// @TEST-ASSERT
AssertTrue(Condition := equal, Message := 'Did not convert DINT to REAL correctly');
AssertTrue(Condition := converted, Message := 'Did not report DINT to REAL conversion was successful');

TEST_FINISHED();
END_METHOD

METHOD PUBLIC Check_DINT_TO_REAL_Max
VAR
	value : DINT := DatatypeLimits.DINT_MAX_VALUE;
	actual : REAL;
	converted : BOOL;
	equal : BOOL;
END_VAR
TEST('Check_DINT_TO_REAL_Max');

// @TEST-RUN
converted := TryConvert_DINT_TO_Destination(value, actual);
equal := actual = DINT_TO_REAL(value);

// @TEST-ASSERT
AssertTrue(Condition := equal, Message := 'Did not convert DINT to REAL correctly');
AssertTrue(Condition := converted, Message := 'Did not report DINT to REAL conversion was successful');

TEST_FINISHED();
END_METHOD

METHOD PUBLIC Check_DINT_TO_SINT_Min
VAR
	value : DINT := DatatypeLimits.MIN_VALUE_OF_DINT_WHICH_CAN_BE_HELD_IN_A_SINT;
	actual : SINT;
	converted : BOOL;
	equal : BOOL;
END_VAR
TEST('Check_DINT_TO_SINT_Min');

// @TEST-RUN
converted := TryConvert_DINT_TO_Destination(value, actual);
equal := actual = DINT_TO_SINT(value);

// @TEST-ASSERT
AssertTrue(Condition := equal, Message := 'Did not convert DINT to SINT correctly');
AssertTrue(Condition := converted, Message := 'Did not report DINT to SINT conversion was successful');

TEST_FINISHED();
END_METHOD

METHOD PUBLIC Check_DINT_TO_SINT_TooHigh
VAR
	value : DINT := DatatypeLimits.DINT_MAX_VALUE;
	actual : SINT;
	converted : BOOL;
END_VAR
TEST('Check_DINT_TO_SINT_TooHigh');

// @TEST-RUN
converted := TryConvert_DINT_TO_Destination(value, actual);

// @TEST-ASSERT
AssertFalse(Condition := converted, Message := 'Did not report DINT to SINT conversion was prevented');

TEST_FINISHED();
END_METHOD

METHOD PUBLIC Check_DINT_TO_SINT_TooLow
VAR
	value : DINT := DatatypeLimits.DINT_MIN_VALUE;
	actual : SINT;
	converted : BOOL;
END_VAR
TEST('Check_DINT_TO_SINT_TooLow');

// @TEST-RUN
converted := TryConvert_DINT_TO_Destination(value, actual);

// @TEST-ASSERT
AssertFalse(Condition := converted, Message := 'Did not report DINT to SINT conversion was prevented');

TEST_FINISHED();
END_METHOD

METHOD PUBLIC Check_DINT_TO_SINT_Max
VAR
	value : DINT := DatatypeLimits.MAX_VALUE_OF_DINT_WHICH_CAN_BE_HELD_IN_A_SINT;
	actual : SINT;
	converted : BOOL;
	equal : BOOL;
END_VAR
TEST('Check_DINT_TO_SINT_Max');

// @TEST-RUN
converted := TryConvert_DINT_TO_Destination(value, actual);
equal := actual = DINT_TO_SINT(value);

// @TEST-ASSERT
AssertTrue(Condition := equal, Message := 'Did not convert DINT to SINT correctly');
AssertTrue(Condition := converted, Message := 'Did not report DINT to SINT conversion was successful');

TEST_FINISHED();
END_METHOD

METHOD PUBLIC Check_DINT_TO_STRING_Min
VAR
	value : DINT := DatatypeLimits.DINT_MIN_VALUE;
	actual : STRING;
	converted : BOOL;
	equal : BOOL;
END_VAR
TEST('Check_DINT_TO_STRING_Min');

// @TEST-RUN
converted := TryConvert_DINT_TO_Destination(value, actual);
equal := actual = DINT_TO_STRING(value);

// @TEST-ASSERT
AssertTrue(Condition := equal, Message := 'Did not convert DINT to STRING correctly');
AssertTrue(Condition := converted, Message := 'Did not report DINT to STRING conversion was successful');

TEST_FINISHED();
END_METHOD

METHOD PUBLIC Check_DINT_TO_STRING_Max
VAR
	value : DINT := DatatypeLimits.DINT_MAX_VALUE;
	actual : STRING;
	converted : BOOL;
	equal : BOOL;
END_VAR
TEST('Check_DINT_TO_STRING_Max');

// @TEST-RUN
converted := TryConvert_DINT_TO_Destination(value, actual);
equal := actual = DINT_TO_STRING(value);

// @TEST-ASSERT
AssertTrue(Condition := equal, Message := 'Did not convert DINT to STRING correctly');
AssertTrue(Condition := converted, Message := 'Did not report DINT to STRING conversion was successful');

TEST_FINISHED();
END_METHOD

METHOD PUBLIC Check_DINT_TO_TIME_Min
VAR
	value : DINT := DatatypeLimits.MIN_VALUE_OF_DINT_WHICH_CAN_BE_HELD_IN_A_TIME;
	actual : TIME;
	converted : BOOL;
	equal : BOOL;
END_VAR
TEST('Check_DINT_TO_TIME_Min');

// @TEST-RUN
converted := TryConvert_DINT_TO_Destination(value, actual);
equal := actual = DINT_TO_TIME(value);

// @TEST-ASSERT
AssertTrue(Condition := equal, Message := 'Did not convert DINT to TIME correctly');
AssertTrue(Condition := converted, Message := 'Did not report DINT to TIME conversion was successful');

TEST_FINISHED();
END_METHOD

METHOD PUBLIC Check_DINT_TO_TIME_TooLow
VAR
	value : DINT := DatatypeLimits.DINT_MIN_VALUE;
	actual : TIME;
	converted : BOOL;
END_VAR
TEST('Check_DINT_TO_TIME_TooLow');

// @TEST-RUN
converted := TryConvert_DINT_TO_Destination(value, actual);

// @TEST-ASSERT
AssertFalse(Condition := converted, Message := 'Did not report DINT to TIME conversion was prevented');

TEST_FINISHED();
END_METHOD

METHOD PUBLIC Check_DINT_TO_TIME_Max
VAR
	value : DINT := DatatypeLimits.DINT_MAX_VALUE;
	actual : TIME;
	converted : BOOL;
	equal : BOOL;
END_VAR
TEST('Check_DINT_TO_TIME_Max');

// @TEST-RUN
converted := TryConvert_DINT_TO_Destination(value, actual);
equal := actual = DINT_TO_TIME(value);

// @TEST-ASSERT
AssertTrue(Condition := equal, Message := 'Did not convert DINT to TIME correctly');
AssertTrue(Condition := converted, Message := 'Did not report DINT to TIME conversion was successful');

TEST_FINISHED();
END_METHOD

METHOD PUBLIC Check_DINT_TO_TOD_Min
VAR
	value : DINT := DatatypeLimits.MIN_VALUE_OF_DINT_WHICH_CAN_BE_HELD_IN_A_TOD;
	actual : TOD;
	converted : BOOL;
	equal : BOOL;
END_VAR
TEST('Check_DINT_TO_TOD_Min');

// @TEST-RUN
converted := TryConvert_DINT_TO_Destination(value, actual);
equal := actual = DINT_TO_TOD(value);

// @TEST-ASSERT
AssertTrue(Condition := equal, Message := 'Did not convert DINT to TOD correctly');
AssertTrue(Condition := converted, Message := 'Did not report DINT to TOD conversion was successful');

TEST_FINISHED();
END_METHOD

METHOD PUBLIC Check_DINT_TO_TOD_TooHigh
VAR
	value : DINT := DatatypeLimits.DINT_MAX_VALUE;
	actual : TOD;
	converted : BOOL;
END_VAR
TEST('Check_DINT_TO_TOD_TooHigh');

// @TEST-RUN
converted := TryConvert_DINT_TO_Destination(value, actual);

// @TEST-ASSERT
AssertFalse(Condition := converted, Message := 'Did not report DINT to TOD conversion was prevented');

TEST_FINISHED();
END_METHOD

METHOD PUBLIC Check_DINT_TO_TOD_TooLow
VAR
	value : DINT := DatatypeLimits.DINT_MIN_VALUE;
	actual : TOD;
	converted : BOOL;
END_VAR
TEST('Check_DINT_TO_TOD_TooLow');

// @TEST-RUN
converted := TryConvert_DINT_TO_Destination(value, actual);

// @TEST-ASSERT
AssertFalse(Condition := converted, Message := 'Did not report DINT to TOD conversion was prevented');

TEST_FINISHED();
END_METHOD

METHOD PUBLIC Check_DINT_TO_TOD_Max
VAR
	value : DINT := DatatypeLimits.MAX_VALUE_OF_DINT_WHICH_CAN_BE_HELD_IN_A_TOD;
	actual : TOD;
	converted : BOOL;
	equal : BOOL;
END_VAR
TEST('Check_DINT_TO_TOD_Max');

// @TEST-RUN
converted := TryConvert_DINT_TO_Destination(value, actual);
equal := actual = DINT_TO_TOD(value);

// @TEST-ASSERT
AssertTrue(Condition := equal, Message := 'Did not convert DINT to TOD correctly');
AssertTrue(Condition := converted, Message := 'Did not report DINT to TOD conversion was successful');

TEST_FINISHED();
END_METHOD

METHOD PUBLIC Check_DINT_TO_UDINT_Min
VAR
	value : DINT := DatatypeLimits.MIN_VALUE_OF_DINT_WHICH_CAN_BE_HELD_IN_A_UDINT;
	actual : UDINT;
	converted : BOOL;
	equal : BOOL;
END_VAR
TEST('Check_DINT_TO_UDINT_Min');

// @TEST-RUN
converted := TryConvert_DINT_TO_Destination(value, actual);
equal := actual = DINT_TO_UDINT(value);

// @TEST-ASSERT
AssertTrue(Condition := equal, Message := 'Did not convert DINT to UDINT correctly');
AssertTrue(Condition := converted, Message := 'Did not report DINT to UDINT conversion was successful');

TEST_FINISHED();
END_METHOD

METHOD PUBLIC Check_DINT_TO_UDINT_TooLow
VAR
	value : DINT := DatatypeLimits.DINT_MIN_VALUE;
	actual : UDINT;
	converted : BOOL;
END_VAR
TEST('Check_DINT_TO_UDINT_TooLow');

// @TEST-RUN
converted := TryConvert_DINT_TO_Destination(value, actual);

// @TEST-ASSERT
AssertFalse(Condition := converted, Message := 'Did not report DINT to UDINT conversion was prevented');

TEST_FINISHED();
END_METHOD

METHOD PUBLIC Check_DINT_TO_UDINT_Max
VAR
	value : DINT := DatatypeLimits.DINT_MAX_VALUE;
	actual : UDINT;
	converted : BOOL;
	equal : BOOL;
END_VAR
TEST('Check_DINT_TO_UDINT_Max');

// @TEST-RUN
converted := TryConvert_DINT_TO_Destination(value, actual);
equal := actual = DINT_TO_UDINT(value);

// @TEST-ASSERT
AssertTrue(Condition := equal, Message := 'Did not convert DINT to UDINT correctly');
AssertTrue(Condition := converted, Message := 'Did not report DINT to UDINT conversion was successful');

TEST_FINISHED();
END_METHOD

METHOD PUBLIC Check_DINT_TO_UINT_Min
VAR
	value : DINT := DatatypeLimits.MIN_VALUE_OF_DINT_WHICH_CAN_BE_HELD_IN_A_UINT;
	actual : UINT;
	converted : BOOL;
	equal : BOOL;
END_VAR
TEST('Check_DINT_TO_UINT_Min');

// @TEST-RUN
converted := TryConvert_DINT_TO_Destination(value, actual);
equal := actual = DINT_TO_UINT(value);

// @TEST-ASSERT
AssertTrue(Condition := equal, Message := 'Did not convert DINT to UINT correctly');
AssertTrue(Condition := converted, Message := 'Did not report DINT to UINT conversion was successful');

TEST_FINISHED();
END_METHOD

METHOD PUBLIC Check_DINT_TO_UINT_TooHigh
VAR
	value : DINT := DatatypeLimits.DINT_MAX_VALUE;
	actual : UINT;
	converted : BOOL;
END_VAR
TEST('Check_DINT_TO_UINT_TooHigh');

// @TEST-RUN
converted := TryConvert_DINT_TO_Destination(value, actual);

// @TEST-ASSERT
AssertFalse(Condition := converted, Message := 'Did not report DINT to UINT conversion was prevented');

TEST_FINISHED();
END_METHOD

METHOD PUBLIC Check_DINT_TO_UINT_TooLow
VAR
	value : DINT := DatatypeLimits.DINT_MIN_VALUE;
	actual : UINT;
	converted : BOOL;
END_VAR
TEST('Check_DINT_TO_UINT_TooLow');

// @TEST-RUN
converted := TryConvert_DINT_TO_Destination(value, actual);

// @TEST-ASSERT
AssertFalse(Condition := converted, Message := 'Did not report DINT to UINT conversion was prevented');

TEST_FINISHED();
END_METHOD

METHOD PUBLIC Check_DINT_TO_UINT_Max
VAR
	value : DINT := DatatypeLimits.MAX_VALUE_OF_DINT_WHICH_CAN_BE_HELD_IN_A_UINT;
	actual : UINT;
	converted : BOOL;
	equal : BOOL;
END_VAR
TEST('Check_DINT_TO_UINT_Max');

// @TEST-RUN
converted := TryConvert_DINT_TO_Destination(value, actual);
equal := actual = DINT_TO_UINT(value);

// @TEST-ASSERT
AssertTrue(Condition := equal, Message := 'Did not convert DINT to UINT correctly');
AssertTrue(Condition := converted, Message := 'Did not report DINT to UINT conversion was successful');

TEST_FINISHED();
END_METHOD

METHOD PUBLIC Check_DINT_TO_ULINT_Min
VAR
	value : DINT := DatatypeLimits.MIN_VALUE_OF_DINT_WHICH_CAN_BE_HELD_IN_A_ULINT;
	actual : ULINT;
	converted : BOOL;
	equal : BOOL;
END_VAR
TEST('Check_DINT_TO_ULINT_Min');

// @TEST-RUN
converted := TryConvert_DINT_TO_Destination(value, actual);
equal := actual = DINT_TO_ULINT(value);

// @TEST-ASSERT
AssertTrue(Condition := equal, Message := 'Did not convert DINT to ULINT correctly');
AssertTrue(Condition := converted, Message := 'Did not report DINT to ULINT conversion was successful');

TEST_FINISHED();
END_METHOD

METHOD PUBLIC Check_DINT_TO_ULINT_TooLow
VAR
	value : DINT := DatatypeLimits.DINT_MIN_VALUE;
	actual : ULINT;
	converted : BOOL;
END_VAR
TEST('Check_DINT_TO_ULINT_TooLow');

// @TEST-RUN
converted := TryConvert_DINT_TO_Destination(value, actual);

// @TEST-ASSERT
AssertFalse(Condition := converted, Message := 'Did not report DINT to ULINT conversion was prevented');

TEST_FINISHED();
END_METHOD

METHOD PUBLIC Check_DINT_TO_ULINT_Max
VAR
	value : DINT := DatatypeLimits.DINT_MAX_VALUE;
	actual : ULINT;
	converted : BOOL;
	equal : BOOL;
END_VAR
TEST('Check_DINT_TO_ULINT_Max');

// @TEST-RUN
converted := TryConvert_DINT_TO_Destination(value, actual);
equal := actual = DINT_TO_ULINT(value);

// @TEST-ASSERT
AssertTrue(Condition := equal, Message := 'Did not convert DINT to ULINT correctly');
AssertTrue(Condition := converted, Message := 'Did not report DINT to ULINT conversion was successful');

TEST_FINISHED();
END_METHOD

METHOD PUBLIC Check_DINT_TO_USINT_Min
VAR
	value : DINT := DatatypeLimits.MIN_VALUE_OF_DINT_WHICH_CAN_BE_HELD_IN_A_USINT;
	actual : USINT;
	converted : BOOL;
	equal : BOOL;
END_VAR
TEST('Check_DINT_TO_USINT_Min');

// @TEST-RUN
converted := TryConvert_DINT_TO_Destination(value, actual);
equal := actual = DINT_TO_USINT(value);

// @TEST-ASSERT
AssertTrue(Condition := equal, Message := 'Did not convert DINT to USINT correctly');
AssertTrue(Condition := converted, Message := 'Did not report DINT to USINT conversion was successful');

TEST_FINISHED();
END_METHOD

METHOD PUBLIC Check_DINT_TO_USINT_TooHigh
VAR
	value : DINT := DatatypeLimits.DINT_MAX_VALUE;
	actual : USINT;
	converted : BOOL;
END_VAR
TEST('Check_DINT_TO_USINT_TooHigh');

// @TEST-RUN
converted := TryConvert_DINT_TO_Destination(value, actual);

// @TEST-ASSERT
AssertFalse(Condition := converted, Message := 'Did not report DINT to USINT conversion was prevented');

TEST_FINISHED();
END_METHOD

METHOD PUBLIC Check_DINT_TO_USINT_TooLow
VAR
	value : DINT := DatatypeLimits.DINT_MIN_VALUE;
	actual : USINT;
	converted : BOOL;
END_VAR
TEST('Check_DINT_TO_USINT_TooLow');

// @TEST-RUN
converted := TryConvert_DINT_TO_Destination(value, actual);

// @TEST-ASSERT
AssertFalse(Condition := converted, Message := 'Did not report DINT to USINT conversion was prevented');

TEST_FINISHED();
END_METHOD

METHOD PUBLIC Check_DINT_TO_USINT_Max
VAR
	value : DINT := DatatypeLimits.MAX_VALUE_OF_DINT_WHICH_CAN_BE_HELD_IN_A_USINT;
	actual : USINT;
	converted : BOOL;
	equal : BOOL;
END_VAR
TEST('Check_DINT_TO_USINT_Max');

// @TEST-RUN
converted := TryConvert_DINT_TO_Destination(value, actual);
equal := actual = DINT_TO_USINT(value);

// @TEST-ASSERT
AssertTrue(Condition := equal, Message := 'Did not convert DINT to USINT correctly');
AssertTrue(Condition := converted, Message := 'Did not report DINT to USINT conversion was successful');

TEST_FINISHED();
END_METHOD

METHOD PUBLIC Check_DINT_TO_WORD_Min
VAR
	value : DINT := DatatypeLimits.MIN_VALUE_OF_DINT_WHICH_CAN_BE_HELD_IN_A_WORD;
	actual : WORD;
	converted : BOOL;
	equal : BOOL;
END_VAR
TEST('Check_DINT_TO_WORD_Min');

// @TEST-RUN
converted := TryConvert_DINT_TO_Destination(value, actual);
equal := actual = DINT_TO_WORD(value);

// @TEST-ASSERT
AssertTrue(Condition := equal, Message := 'Did not convert DINT to WORD correctly');
AssertTrue(Condition := converted, Message := 'Did not report DINT to WORD conversion was successful');

TEST_FINISHED();
END_METHOD

METHOD PUBLIC Check_DINT_TO_WORD_TooHigh
VAR
	value : DINT := DatatypeLimits.DINT_MAX_VALUE;
	actual : WORD;
	converted : BOOL;
END_VAR
TEST('Check_DINT_TO_WORD_TooHigh');

// @TEST-RUN
converted := TryConvert_DINT_TO_Destination(value, actual);

// @TEST-ASSERT
AssertFalse(Condition := converted, Message := 'Did not report DINT to WORD conversion was prevented');

TEST_FINISHED();
END_METHOD

METHOD PUBLIC Check_DINT_TO_WORD_TooLow
VAR
	value : DINT := DatatypeLimits.DINT_MIN_VALUE;
	actual : WORD;
	converted : BOOL;
END_VAR
TEST('Check_DINT_TO_WORD_TooLow');

// @TEST-RUN
converted := TryConvert_DINT_TO_Destination(value, actual);

// @TEST-ASSERT
AssertFalse(Condition := converted, Message := 'Did not report DINT to WORD conversion was prevented');

TEST_FINISHED();
END_METHOD

METHOD PUBLIC Check_DINT_TO_WORD_Max
VAR
	value : DINT := DatatypeLimits.MAX_VALUE_OF_DINT_WHICH_CAN_BE_HELD_IN_A_WORD;
	actual : WORD;
	converted : BOOL;
	equal : BOOL;
END_VAR
TEST('Check_DINT_TO_WORD_Max');

// @TEST-RUN
converted := TryConvert_DINT_TO_Destination(value, actual);
equal := actual = DINT_TO_WORD(value);

// @TEST-ASSERT
AssertTrue(Condition := equal, Message := 'Did not convert DINT to WORD correctly');
AssertTrue(Condition := converted, Message := 'Did not report DINT to WORD conversion was successful');

TEST_FINISHED();
END_METHOD

END_FUNCTION_BLOCK

// ---- Tests/LINT_TO_TestSuite.TcPOU
FUNCTION_BLOCK PUBLIC LINT_TO_TestSuite EXTENDS TcUnit.FB_TestSuite
VAR
END_VAR

Check_LINT_TO_BOOL_Max();
Check_LINT_TO_BOOL_Min();
Check_LINT_TO_BYTE_Max();
Check_LINT_TO_BYTE_Min();
Check_LINT_TO_BYTE_TooHigh();
Check_LINT_TO_BYTE_TooLow();
Check_LINT_TO_WORD_Max();
Check_LINT_TO_WORD_Min();
Check_LINT_TO_WORD_TooHigh();
Check_LINT_TO_WORD_TooLow();
Check_LINT_TO_DWORD_Max();
Check_LINT_TO_DWORD_Min();
Check_LINT_TO_DWORD_TooHigh();
Check_LINT_TO_DWORD_TooLow();
Check_LINT_TO_LWORD_Max();
Check_LINT_TO_LWORD_Min();
Check_LINT_TO_LWORD_TooLow();
Check_LINT_TO_SINT_Max();
Check_LINT_TO_SINT_Min();
Check_LINT_TO_SINT_TooHigh();
Check_LINT_TO_SINT_TooLow();
Check_LINT_TO_INT_Max();
Check_LINT_TO_INT_Min();
Check_LINT_TO_INT_TooHigh();
Check_LINT_TO_INT_TooLow();
Check_LINT_TO_DINT_Max();
Check_LINT_TO_DINT_Min();
Check_LINT_TO_DINT_TooHigh();
Check_LINT_TO_DINT_TooLow();
Check_LINT_TO_LINT_Max();
Check_LINT_TO_LINT_Min();
Check_LINT_TO_USINT_Max();
Check_LINT_TO_USINT_Min();
Check_LINT_TO_USINT_TooHigh();
Check_LINT_TO_USINT_TooLow();
Check_LINT_TO_UINT_Max();
Check_LINT_TO_UINT_Min();
Check_LINT_TO_UINT_TooHigh();
Check_LINT_TO_UINT_TooLow();
Check_LINT_TO_UDINT_Max();
Check_LINT_TO_UDINT_Min();
Check_LINT_TO_UDINT_TooHigh();
Check_LINT_TO_UDINT_TooLow();
Check_LINT_TO_ULINT_Max();
Check_LINT_TO_ULINT_Min();
Check_LINT_TO_ULINT_TooLow();
Check_LINT_TO_REAL_Max();
Check_LINT_TO_REAL_Min();
Check_LINT_TO_LREAL_Max();
Check_LINT_TO_LREAL_Min();
Check_LINT_TO_TIME_Max();
Check_LINT_TO_TIME_Min();
Check_LINT_TO_TIME_TooHigh();
Check_LINT_TO_TIME_TooLow();
Check_LINT_TO_TOD_Max();
Check_LINT_TO_TOD_Min();
Check_LINT_TO_TOD_TooHigh();
Check_LINT_TO_TOD_TooLow();
Check_LINT_TO_DATE_Max();
Check_LINT_TO_DATE_Min();
Check_LINT_TO_DATE_TooHigh();
Check_LINT_TO_DATE_TooLow();
Check_LINT_TO_DT_Max();
Check_LINT_TO_DT_Min();
Check_LINT_TO_DT_TooHigh();
Check_LINT_TO_DT_TooLow();
Check_LINT_TO_STRING_Max();
Check_LINT_TO_STRING_Min();

METHOD PUBLIC Check_LINT_TO_BOOL_Min
VAR
	value : LINT := DatatypeLimits.LINT_MIN_VALUE;
	actual : BOOL;
	converted : BOOL;
	equal : BOOL;
END_VAR
TEST('Check_LINT_TO_BOOL_Min');

// @TEST-RUN
converted := TryConvert_LINT_TO_Destination(value, actual);
equal := actual = LINT_TO_BOOL(value);

// @TEST-ASSERT
AssertTrue(Condition := equal, Message := 'Did not convert LINT to BOOL correctly');
AssertTrue(Condition := converted, Message := 'Did not report LINT to BOOL conversion was successful');

TEST_FINISHED();
END_METHOD

METHOD PUBLIC Check_LINT_TO_BOOL_Max
VAR
	value : LINT := DatatypeLimits.LINT_MAX_VALUE;
	actual : BOOL;
	converted : BOOL;
	equal : BOOL;
END_VAR
TEST('Check_LINT_TO_BOOL_Max');

// @TEST-RUN
converted := TryConvert_LINT_TO_Destination(value, actual);
equal := actual = LINT_TO_BOOL(value);

// @TEST-ASSERT
AssertTrue(Condition := equal, Message := 'Did not convert LINT to BOOL correctly');
AssertTrue(Condition := converted, Message := 'Did not report LINT to BOOL conversion was successful');

TEST_FINISHED();
END_METHOD

METHOD PUBLIC Check_LINT_TO_BYTE_Min
VAR
	value : LINT := DatatypeLimits.MIN_VALUE_OF_LINT_WHICH_CAN_BE_HELD_IN_A_BYTE;
	actual : BYTE;
	converted : BOOL;
	equal : BOOL;
END_VAR
TEST('Check_LINT_TO_BYTE_Min');

// @TEST-RUN
converted := TryConvert_LINT_TO_Destination(value, actual);
equal := actual = LINT_TO_BYTE(value);

// @TEST-ASSERT
AssertTrue(Condition := equal, Message := 'Did not convert LINT to BYTE correctly');
AssertTrue(Condition := converted, Message := 'Did not report LINT to BYTE conversion was successful');

TEST_FINISHED();
END_METHOD

METHOD PUBLIC Check_LINT_TO_BYTE_TooHigh
VAR
	value : LINT := DatatypeLimits.LINT_MAX_VALUE;
	actual : BYTE;
	converted : BOOL;
END_VAR
TEST('Check_LINT_TO_BYTE_TooHigh');

// @TEST-RUN
converted := TryConvert_LINT_TO_Destination(value, actual);

// @TEST-ASSERT
AssertFalse(Condition := converted, Message := 'Did not report LINT to BYTE conversion was prevented');

TEST_FINISHED();
END_METHOD

METHOD PUBLIC Check_LINT_TO_BYTE_TooLow
VAR
	value : LINT := DatatypeLimits.LINT_MIN_VALUE;
	actual : BYTE;
	converted : BOOL;
END_VAR
TEST('Check_LINT_TO_BYTE_TooLow');

// @TEST-RUN
converted := TryConvert_LINT_TO_Destination(value, actual);

// @TEST-ASSERT
AssertFalse(Condition := converted, Message := 'Did not report LINT to BYTE conversion was prevented');

TEST_FINISHED();
END_METHOD

METHOD PUBLIC Check_LINT_TO_BYTE_Max
VAR
	value : LINT := DatatypeLimits.MAX_VALUE_OF_LINT_WHICH_CAN_BE_HELD_IN_A_BYTE;
	actual : BYTE;
	converted : BOOL;
	equal : BOOL;
END_VAR
TEST('Check_LINT_TO_BYTE_Max');

// @TEST-RUN
converted := TryConvert_LINT_TO_Destination(value, actual);
equal := actual = LINT_TO_BYTE(value);

// @TEST-ASSERT
AssertTrue(Condition := equal, Message := 'Did not convert LINT to BYTE correctly');
AssertTrue(Condition := converted, Message := 'Did not report LINT to BYTE conversion was successful');

TEST_FINISHED();
END_METHOD

METHOD PUBLIC Check_LINT_TO_DATE_Min
VAR
	value : LINT := DatatypeLimits.MIN_VALUE_OF_LINT_WHICH_CAN_BE_HELD_IN_A_DATE;
	actual : DATE;
	converted : BOOL;
	equal : BOOL;
END_VAR
TEST('Check_LINT_TO_DATE_Min');

// @TEST-RUN
converted := TryConvert_LINT_TO_Destination(value, actual);
equal := actual = LINT_TO_DATE(value);

// @TEST-ASSERT
AssertTrue(Condition := equal, Message := 'Did not convert LINT to DATE correctly');
AssertTrue(Condition := converted, Message := 'Did not report LINT to DATE conversion was successful');

TEST_FINISHED();
END_METHOD

METHOD PUBLIC Check_LINT_TO_DATE_TooHigh
VAR
	value : LINT := DatatypeLimits.LINT_MAX_VALUE;
	actual : DATE;
	converted : BOOL;
END_VAR
TEST('Check_LINT_TO_DATE_TooHigh');

// @TEST-RUN
converted := TryConvert_LINT_TO_Destination(value, actual);

// @TEST-ASSERT
AssertFalse(Condition := converted, Message := 'Did not report LINT to DATE conversion was prevented');

TEST_FINISHED();
END_METHOD

METHOD PUBLIC Check_LINT_TO_DATE_TooLow
VAR
	value : LINT := DatatypeLimits.LINT_MIN_VALUE;
	actual : DATE;
	converted : BOOL;
END_VAR
TEST('Check_LINT_TO_DATE_TooLow');

// @TEST-RUN
converted := TryConvert_LINT_TO_Destination(value, actual);

// @TEST-ASSERT
AssertFalse(Condition := converted, Message := 'Did not report LINT to DATE conversion was prevented');

TEST_FINISHED();
END_METHOD

METHOD PUBLIC Check_LINT_TO_DATE_Max
VAR
	value : LINT := DatatypeLimits.MAX_VALUE_OF_LINT_WHICH_CAN_BE_HELD_IN_A_DATE;
	actual : DATE;
	converted : BOOL;
	equal : BOOL;
END_VAR
TEST('Check_LINT_TO_DATE_Max');

// @TEST-RUN
converted := TryConvert_LINT_TO_Destination(value, actual);
equal := actual = LINT_TO_DATE(value);

// @TEST-ASSERT
AssertTrue(Condition := equal, Message := 'Did not convert LINT to DATE correctly');
AssertTrue(Condition := converted, Message := 'Did not report LINT to DATE conversion was successful');

TEST_FINISHED();
END_METHOD

METHOD PUBLIC Check_LINT_TO_DINT_Min
VAR
	value : LINT := DatatypeLimits.MIN_VALUE_OF_LINT_WHICH_CAN_BE_HELD_IN_A_DINT;
	actual : DINT;
	converted : BOOL;
	equal : BOOL;
END_VAR
TEST('Check_LINT_TO_DINT_Min');

// @TEST-RUN
converted := TryConvert_LINT_TO_Destination(value, actual);
equal := actual = LINT_TO_DINT(value);

// @TEST-ASSERT
AssertTrue(Condition := equal, Message := 'Did not convert LINT to DINT correctly');
AssertTrue(Condition := converted, Message := 'Did not report LINT to DINT conversion was successful');

TEST_FINISHED();
END_METHOD

METHOD PUBLIC Check_LINT_TO_DINT_TooHigh
VAR
	value : LINT := DatatypeLimits.LINT_MAX_VALUE;
	actual : DINT;
	converted : BOOL;
END_VAR
TEST('Check_LINT_TO_DINT_TooHigh');

// @TEST-RUN
converted := TryConvert_LINT_TO_Destination(value, actual);

// @TEST-ASSERT
AssertFalse(Condition := converted, Message := 'Did not report LINT to DINT conversion was prevented');

TEST_FINISHED();
END_METHOD

METHOD PUBLIC Check_LINT_TO_DINT_TooLow
VAR
	value : LINT := DatatypeLimits.LINT_MIN_VALUE;
	actual : DINT;
	converted : BOOL;
END_VAR
TEST('Check_LINT_TO_DINT_TooLow');

// @TEST-RUN
converted := TryConvert_LINT_TO_Destination(value, actual);

// @TEST-ASSERT
AssertFalse(Condition := converted, Message := 'Did not report LINT to DINT conversion was prevented');

TEST_FINISHED();
END_METHOD

METHOD PUBLIC Check_LINT_TO_DINT_Max
VAR
	value : LINT := DatatypeLimits.MAX_VALUE_OF_LINT_WHICH_CAN_BE_HELD_IN_A_DINT;
	actual : DINT;
	converted : BOOL;
	equal : BOOL;
END_VAR
TEST('Check_LINT_TO_DINT_Max');

// @TEST-RUN
converted := TryConvert_LINT_TO_Destination(value, actual);
equal := actual = LINT_TO_DINT(value);

// @TEST-ASSERT
AssertTrue(Condition := equal, Message := 'Did not convert LINT to DINT correctly');
AssertTrue(Condition := converted, Message := 'Did not report LINT to DINT conversion was successful');

TEST_FINISHED();
END_METHOD

METHOD PUBLIC Check_LINT_TO_DT_Min
VAR
	value : LINT := DatatypeLimits.MIN_VALUE_OF_LINT_WHICH_CAN_BE_HELD_IN_A_DT;
	actual : DT;
	converted : BOOL;
	equal : BOOL;
END_VAR
TEST('Check_LINT_TO_DT_Min');

// @TEST-RUN
converted := TryConvert_LINT_TO_Destination(value, actual);
equal := actual = LINT_TO_DT(value);

// @TEST-ASSERT
AssertTrue(Condition := equal, Message := 'Did not convert LINT to DT correctly');
AssertTrue(Condition := converted, Message := 'Did not report LINT to DT conversion was successful');

TEST_FINISHED();
END_METHOD

METHOD PUBLIC Check_LINT_TO_DT_TooHigh
VAR
	value : LINT := DatatypeLimits.LINT_MAX_VALUE;
	actual : DT;
	converted : BOOL;
END_VAR
TEST('Check_LINT_TO_DT_TooHigh');

// @TEST-RUN
converted := TryConvert_LINT_TO_Destination(value, actual);

// @TEST-ASSERT
AssertFalse(Condition := converted, Message := 'Did not report LINT to DT conversion was prevented');

TEST_FINISHED();
END_METHOD

METHOD PUBLIC Check_LINT_TO_DT_TooLow
VAR
	value : LINT := DatatypeLimits.LINT_MIN_VALUE;
	actual : DT;
	converted : BOOL;
END_VAR
TEST('Check_LINT_TO_DT_TooLow');

// @TEST-RUN
converted := TryConvert_LINT_TO_Destination(value, actual);

// @TEST-ASSERT
AssertFalse(Condition := converted, Message := 'Did not report LINT to DT conversion was prevented');

TEST_FINISHED();
END_METHOD

METHOD PUBLIC Check_LINT_TO_DT_Max
VAR
	value : LINT := DatatypeLimits.MAX_VALUE_OF_LINT_WHICH_CAN_BE_HELD_IN_A_DT;
	actual : DT;
	converted : BOOL;
	equal : BOOL;
END_VAR
TEST('Check_LINT_TO_DT_Max');

// @TEST-RUN
converted := TryConvert_LINT_TO_Destination(value, actual);
equal := actual = LINT_TO_DT(value);

// @TEST-ASSERT
AssertTrue(Condition := equal, Message := 'Did not convert LINT to DT correctly');
AssertTrue(Condition := converted, Message := 'Did not report LINT to DT conversion was successful');

TEST_FINISHED();
END_METHOD

METHOD PUBLIC Check_LINT_TO_DWORD_Min
VAR
	value : LINT := DatatypeLimits.MIN_VALUE_OF_LINT_WHICH_CAN_BE_HELD_IN_A_DWORD;
	actual : DWORD;
	converted : BOOL;
	equal : BOOL;
END_VAR
TEST('Check_LINT_TO_DWORD_Min');

// @TEST-RUN
converted := TryConvert_LINT_TO_Destination(value, actual);
equal := actual = LINT_TO_DWORD(value);

// @TEST-ASSERT
AssertTrue(Condition := equal, Message := 'Did not convert LINT to DWORD correctly');
AssertTrue(Condition := converted, Message := 'Did not report LINT to DWORD conversion was successful');

TEST_FINISHED();
END_METHOD

METHOD PUBLIC Check_LINT_TO_DWORD_TooHigh
VAR
	value : LINT := DatatypeLimits.LINT_MAX_VALUE;
	actual : DWORD;
	converted : BOOL;
END_VAR
TEST('Check_LINT_TO_DWORD_TooHigh');

// @TEST-RUN
converted := TryConvert_LINT_TO_Destination(value, actual);

// @TEST-ASSERT
AssertFalse(Condition := converted, Message := 'Did not report LINT to DWORD conversion was prevented');

TEST_FINISHED();
END_METHOD

METHOD PUBLIC Check_LINT_TO_DWORD_TooLow
VAR
	value : LINT := DatatypeLimits.LINT_MIN_VALUE;
	actual : DWORD;
	converted : BOOL;
END_VAR
TEST('Check_LINT_TO_DWORD_TooLow');

// @TEST-RUN
converted := TryConvert_LINT_TO_Destination(value, actual);

// @TEST-ASSERT
AssertFalse(Condition := converted, Message := 'Did not report LINT to DWORD conversion was prevented');

TEST_FINISHED();
END_METHOD

METHOD PUBLIC Check_LINT_TO_DWORD_Max
VAR
	value : LINT := DatatypeLimits.MAX_VALUE_OF_LINT_WHICH_CAN_BE_HELD_IN_A_DWORD;
	actual : DWORD;
	converted : BOOL;
	equal : BOOL;
END_VAR
TEST('Check_LINT_TO_DWORD_Max');

// @TEST-RUN
converted := TryConvert_LINT_TO_Destination(value, actual);
equal := actual = LINT_TO_DWORD(value);

// @TEST-ASSERT
AssertTrue(Condition := equal, Message := 'Did not convert LINT to DWORD correctly');
AssertTrue(Condition := converted, Message := 'Did not report LINT to DWORD conversion was successful');

TEST_FINISHED();
END_METHOD

METHOD PUBLIC Check_LINT_TO_INT_Min
VAR
	value : LINT := DatatypeLimits.MIN_VALUE_OF_LINT_WHICH_CAN_BE_HELD_IN_A_INT;
	actual : INT;
	converted : BOOL;
	equal : BOOL;
END_VAR
TEST('Check_LINT_TO_INT_Min');

// @TEST-RUN
converted := TryConvert_LINT_TO_Destination(value, actual);
equal := actual = LINT_TO_INT(value);

// @TEST-ASSERT
AssertTrue(Condition := equal, Message := 'Did not convert LINT to INT correctly');
AssertTrue(Condition := converted, Message := 'Did not report LINT to INT conversion was successful');

TEST_FINISHED();
END_METHOD

METHOD PUBLIC Check_LINT_TO_INT_TooHigh
VAR
	value : LINT := DatatypeLimits.LINT_MAX_VALUE;
	actual : INT;
	converted : BOOL;
END_VAR
TEST('Check_LINT_TO_INT_TooHigh');

// @TEST-RUN
converted := TryConvert_LINT_TO_Destination(value, actual);

// @TEST-ASSERT
AssertFalse(Condition := converted, Message := 'Did not report LINT to INT conversion was prevented');

TEST_FINISHED();
END_METHOD

METHOD PUBLIC Check_LINT_TO_INT_TooLow
VAR
	value : LINT := DatatypeLimits.LINT_MIN_VALUE;
	actual : INT;
	converted : BOOL;
END_VAR
TEST('Check_LINT_TO_INT_TooLow');

// @TEST-RUN
converted := TryConvert_LINT_TO_Destination(value, actual);

// @TEST-ASSERT
AssertFalse(Condition := converted, Message := 'Did not report LINT to INT conversion was prevented');

TEST_FINISHED();
END_METHOD

METHOD PUBLIC Check_LINT_TO_INT_Max
VAR
	value : LINT := DatatypeLimits.MAX_VALUE_OF_LINT_WHICH_CAN_BE_HELD_IN_A_INT;
	actual : INT;
	converted : BOOL;
	equal : BOOL;
END_VAR
TEST('Check_LINT_TO_INT_Max');

// @TEST-RUN
converted := TryConvert_LINT_TO_Destination(value, actual);
equal := actual = LINT_TO_INT(value);

// @TEST-ASSERT
AssertTrue(Condition := equal, Message := 'Did not convert LINT to INT correctly');
AssertTrue(Condition := converted, Message := 'Did not report LINT to INT conversion was successful');

TEST_FINISHED();
END_METHOD

METHOD PUBLIC Check_LINT_TO_LINT_Min
VAR
	value : LINT := DatatypeLimits.LINT_MIN_VALUE;
	actual : LINT;
	converted : BOOL;
	equal : BOOL;
END_VAR
TEST('Check_LINT_TO_LINT_Min');

// @TEST-RUN
converted := TryConvert_LINT_TO_Destination(value, actual);
equal := actual = value;

// @TEST-ASSERT
AssertTrue(Condition := equal, Message := 'Did not convert LINT to LINT correctly');
AssertTrue(Condition := converted, Message := 'Did not report LINT to LINT conversion was successful');

TEST_FINISHED();
END_METHOD

METHOD PUBLIC Check_LINT_TO_LINT_Max
VAR
	value : LINT := DatatypeLimits.LINT_MAX_VALUE;
	actual : LINT;
	converted : BOOL;
	equal : BOOL;
END_VAR
TEST('Check_LINT_TO_LINT_Max');

// @TEST-RUN
converted := TryConvert_LINT_TO_Destination(value, actual);
equal := actual = value;

// @TEST-ASSERT
AssertTrue(Condition := equal, Message := 'Did not convert LINT to LINT correctly');
AssertTrue(Condition := converted, Message := 'Did not report LINT to LINT conversion was successful');

TEST_FINISHED();
END_METHOD

METHOD PUBLIC Check_LINT_TO_LREAL_Min
VAR
	value : LINT := DatatypeLimits.LINT_MIN_VALUE;
	actual : LREAL;
	converted : BOOL;
	equal : BOOL;
END_VAR
TEST('Check_LINT_TO_LREAL_Min');

// @TEST-RUN
converted := TryConvert_LINT_TO_Destination(value, actual);
equal := actual = LINT_TO_LREAL(value);

// @TEST-ASSERT
AssertTrue(Condition := equal, Message := 'Did not convert LINT to LREAL correctly');
AssertTrue(Condition := converted, Message := 'Did not report LINT to LREAL conversion was successful');

TEST_FINISHED();
END_METHOD

METHOD PUBLIC Check_LINT_TO_LREAL_Max
VAR
	value : LINT := DatatypeLimits.LINT_MAX_VALUE;
	actual : LREAL;
	converted : BOOL;
	equal : BOOL;
END_VAR
TEST('Check_LINT_TO_LREAL_Max');

// @TEST-RUN
converted := TryConvert_LINT_TO_Destination(value, actual);
equal := actual = LINT_TO_LREAL(value);

// @TEST-ASSERT
AssertTrue(Condition := equal, Message := 'Did not convert LINT to LREAL correctly');
AssertTrue(Condition := converted, Message := 'Did not report LINT to LREAL conversion was successful');

TEST_FINISHED();
END_METHOD

METHOD PUBLIC Check_LINT_TO_LWORD_Min
VAR
	value : LINT := DatatypeLimits.MIN_VALUE_OF_LINT_WHICH_CAN_BE_HELD_IN_A_LWORD;
	actual : LWORD;
	converted : BOOL;
	equal : BOOL;
END_VAR
TEST('Check_LINT_TO_LWORD_Min');

// @TEST-RUN
converted := TryConvert_LINT_TO_Destination(value, actual);
equal := actual = LINT_TO_LWORD(value);

// @TEST-ASSERT
AssertTrue(Condition := equal, Message := 'Did not convert LINT to LWORD correctly');
AssertTrue(Condition := converted, Message := 'Did not report LINT to LWORD conversion was successful');

TEST_FINISHED();
END_METHOD

METHOD PUBLIC Check_LINT_TO_LWORD_TooLow
VAR
	value : LINT := DatatypeLimits.LINT_MIN_VALUE;
	actual : LWORD;
	converted : BOOL;
END_VAR
TEST('Check_LINT_TO_LWORD_TooLow');

// @TEST-RUN
converted := TryConvert_LINT_TO_Destination(value, actual);

// @TEST-ASSERT
AssertFalse(Condition := converted, Message := 'Did not report LINT to LWORD conversion was prevented');

TEST_FINISHED();
END_METHOD

METHOD PUBLIC Check_LINT_TO_LWORD_Max
VAR
	value : LINT := DatatypeLimits.LINT_MAX_VALUE;
	actual : LWORD;
	converted : BOOL;
	equal : BOOL;
END_VAR
TEST('Check_LINT_TO_LWORD_Max');

// @TEST-RUN
converted := TryConvert_LINT_TO_Destination(value, actual);
equal := actual = LINT_TO_LWORD(value);

// @TEST-ASSERT
AssertTrue(Condition := equal, Message := 'Did not convert LINT to LWORD correctly');
AssertTrue(Condition := converted, Message := 'Did not report LINT to LWORD conversion was successful');

TEST_FINISHED();
END_METHOD

METHOD PUBLIC Check_LINT_TO_REAL_Min
VAR
	value : LINT := DatatypeLimits.LINT_MIN_VALUE;
	actual : REAL;
	converted : BOOL;
	equal : BOOL;
END_VAR
TEST('Check_LINT_TO_REAL_Min');

// @TEST-RUN
converted := TryConvert_LINT_TO_Destination(value, actual);
equal := actual = LINT_TO_REAL(value);

// @TEST-ASSERT
AssertTrue(Condition := equal, Message := 'Did not convert LINT to REAL correctly');
AssertTrue(Condition := converted, Message := 'Did not report LINT to REAL conversion was successful');

TEST_FINISHED();
END_METHOD

METHOD PUBLIC Check_LINT_TO_REAL_Max
VAR
	value : LINT := DatatypeLimits.LINT_MAX_VALUE;
	actual : REAL;
	converted : BOOL;
	equal : BOOL;
END_VAR
TEST('Check_LINT_TO_REAL_Max');

// @TEST-RUN
converted := TryConvert_LINT_TO_Destination(value, actual);
equal := actual = LINT_TO_REAL(value);

// @TEST-ASSERT
AssertTrue(Condition := equal, Message := 'Did not convert LINT to REAL correctly');
AssertTrue(Condition := converted, Message := 'Did not report LINT to REAL conversion was successful');

TEST_FINISHED();
END_METHOD

METHOD PUBLIC Check_LINT_TO_SINT_Min
VAR
	value : LINT := DatatypeLimits.MIN_VALUE_OF_LINT_WHICH_CAN_BE_HELD_IN_A_SINT;
	actual : SINT;
	converted : BOOL;
	equal : BOOL;
END_VAR
TEST('Check_LINT_TO_SINT_Min');

// @TEST-RUN
converted := TryConvert_LINT_TO_Destination(value, actual);
equal := actual = LINT_TO_SINT(value);

// @TEST-ASSERT
AssertTrue(Condition := equal, Message := 'Did not convert LINT to SINT correctly');
AssertTrue(Condition := converted, Message := 'Did not report LINT to SINT conversion was successful');

TEST_FINISHED();
END_METHOD

METHOD PUBLIC Check_LINT_TO_SINT_TooHigh
VAR
	value : LINT := DatatypeLimits.LINT_MAX_VALUE;
	actual : SINT;
	converted : BOOL;
END_VAR
TEST('Check_LINT_TO_SINT_TooHigh');

// @TEST-RUN
converted := TryConvert_LINT_TO_Destination(value, actual);

// @TEST-ASSERT
AssertFalse(Condition := converted, Message := 'Did not report LINT to SINT conversion was prevented');

TEST_FINISHED();
END_METHOD

METHOD PUBLIC Check_LINT_TO_SINT_TooLow
VAR
	value : LINT := DatatypeLimits.LINT_MIN_VALUE;
	actual : SINT;
	converted : BOOL;
END_VAR
TEST('Check_LINT_TO_SINT_TooLow');

// @TEST-RUN
converted := TryConvert_LINT_TO_Destination(value, actual);

// @TEST-ASSERT
AssertFalse(Condition := converted, Message := 'Did not report LINT to SINT conversion was prevented');

TEST_FINISHED();
END_METHOD

METHOD PUBLIC Check_LINT_TO_SINT_Max
VAR
	value : LINT := DatatypeLimits.MAX_VALUE_OF_LINT_WHICH_CAN_BE_HELD_IN_A_SINT;
	actual : SINT;
	converted : BOOL;
	equal : BOOL;
END_VAR
TEST('Check_LINT_TO_SINT_Max');

// @TEST-RUN
converted := TryConvert_LINT_TO_Destination(value, actual);
equal := actual = LINT_TO_SINT(value);

// @TEST-ASSERT
AssertTrue(Condition := equal, Message := 'Did not convert LINT to SINT correctly');
AssertTrue(Condition := converted, Message := 'Did not report LINT to SINT conversion was successful');

TEST_FINISHED();
END_METHOD

METHOD PUBLIC Check_LINT_TO_STRING_Min
VAR
	value : LINT := DatatypeLimits.LINT_MIN_VALUE;
	actual : STRING;
	converted : BOOL;
	equal : BOOL;
END_VAR
TEST('Check_LINT_TO_STRING_Min');

// @TEST-RUN
converted := TryConvert_LINT_TO_Destination(value, actual);
equal := actual = LINT_TO_STRING(value);

// @TEST-ASSERT
AssertTrue(Condition := equal, Message := 'Did not convert LINT to STRING correctly');
AssertTrue(Condition := converted, Message := 'Did not report LINT to STRING conversion was successful');

TEST_FINISHED();
END_METHOD

METHOD PUBLIC Check_LINT_TO_STRING_Max
VAR
	value : LINT := DatatypeLimits.LINT_MAX_VALUE;
	actual : STRING;
	converted : BOOL;
	equal : BOOL;
END_VAR
TEST('Check_LINT_TO_STRING_Max');

// @TEST-RUN
converted := TryConvert_LINT_TO_Destination(value, actual);
equal := actual = LINT_TO_STRING(value);

// @TEST-ASSERT
AssertTrue(Condition := equal, Message := 'Did not convert LINT to STRING correctly');
AssertTrue(Condition := converted, Message := 'Did not report LINT to STRING conversion was successful');

TEST_FINISHED();
END_METHOD

METHOD PUBLIC Check_LINT_TO_TIME_Min
VAR
	value : LINT := DatatypeLimits.MIN_VALUE_OF_LINT_WHICH_CAN_BE_HELD_IN_A_TIME;
	actual : TIME;
	converted : BOOL;
	equal : BOOL;
END_VAR
TEST('Check_LINT_TO_TIME_Min');

// @TEST-RUN
converted := TryConvert_LINT_TO_Destination(value, actual);
equal := actual = LINT_TO_TIME(value);

// @TEST-ASSERT
AssertTrue(Condition := equal, Message := 'Did not convert LINT to TIME correctly');
AssertTrue(Condition := converted, Message := 'Did not report LINT to TIME conversion was successful');

TEST_FINISHED();
END_METHOD

METHOD PUBLIC Check_LINT_TO_TIME_TooHigh
VAR
	value : LINT := DatatypeLimits.LINT_MAX_VALUE;
	actual : TIME;
	converted : BOOL;
END_VAR
TEST('Check_LINT_TO_TIME_TooHigh');

// @TEST-RUN
converted := TryConvert_LINT_TO_Destination(value, actual);

// @TEST-ASSERT
AssertFalse(Condition := converted, Message := 'Did not report LINT to TIME conversion was prevented');

TEST_FINISHED();
END_METHOD

METHOD PUBLIC Check_LINT_TO_TIME_TooLow
VAR
	value : LINT := DatatypeLimits.LINT_MIN_VALUE;
	actual : TIME;
	converted : BOOL;
END_VAR
TEST('Check_LINT_TO_TIME_TooLow');

// @TEST-RUN
converted := TryConvert_LINT_TO_Destination(value, actual);

// @TEST-ASSERT
AssertFalse(Condition := converted, Message := 'Did not report LINT to TIME conversion was prevented');

TEST_FINISHED();
END_METHOD

METHOD PUBLIC Check_LINT_TO_TIME_Max
VAR
	value : LINT := DatatypeLimits.MAX_VALUE_OF_LINT_WHICH_CAN_BE_HELD_IN_A_TIME;
	actual : TIME;
	converted : BOOL;
	equal : BOOL;
END_VAR
TEST('Check_LINT_TO_TIME_Max');

// @TEST-RUN
converted := TryConvert_LINT_TO_Destination(value, actual);
equal := actual = LINT_TO_TIME(value);

// @TEST-ASSERT
AssertTrue(Condition := equal, Message := 'Did not convert LINT to TIME correctly');
AssertTrue(Condition := converted, Message := 'Did not report LINT to TIME conversion was successful');

TEST_FINISHED();
END_METHOD

METHOD PUBLIC Check_LINT_TO_TOD_Min
VAR
	value : LINT := DatatypeLimits.MIN_VALUE_OF_LINT_WHICH_CAN_BE_HELD_IN_A_TOD;
	actual : TOD;
	converted : BOOL;
	equal : BOOL;
END_VAR
TEST('Check_LINT_TO_TOD_Min');

// @TEST-RUN
converted := TryConvert_LINT_TO_Destination(value, actual);
equal := actual = LINT_TO_TOD(value);

// @TEST-ASSERT
AssertTrue(Condition := equal, Message := 'Did not convert LINT to TOD correctly');
AssertTrue(Condition := converted, Message := 'Did not report LINT to TOD conversion was successful');

TEST_FINISHED();
END_METHOD

METHOD PUBLIC Check_LINT_TO_TOD_TooHigh
VAR
	value : LINT := DatatypeLimits.LINT_MAX_VALUE;
	actual : TOD;
	converted : BOOL;
END_VAR
TEST('Check_LINT_TO_TOD_TooHigh');

// @TEST-RUN
converted := TryConvert_LINT_TO_Destination(value, actual);

// @TEST-ASSERT
AssertFalse(Condition := converted, Message := 'Did not report LINT to TOD conversion was prevented');

TEST_FINISHED();
END_METHOD

METHOD PUBLIC Check_LINT_TO_TOD_TooLow
VAR
	value : LINT := DatatypeLimits.LINT_MIN_VALUE;
	actual : TOD;
	converted : BOOL;
END_VAR
TEST('Check_LINT_TO_TOD_TooLow');

// @TEST-RUN
converted := TryConvert_LINT_TO_Destination(value, actual);

// @TEST-ASSERT
AssertFalse(Condition := converted, Message := 'Did not report LINT to TOD conversion was prevented');

TEST_FINISHED();
END_METHOD

METHOD PUBLIC Check_LINT_TO_TOD_Max
VAR
	value : LINT := DatatypeLimits.MAX_VALUE_OF_LINT_WHICH_CAN_BE_HELD_IN_A_TOD;
	actual : TOD;
	converted : BOOL;
	equal : BOOL;
END_VAR
TEST('Check_LINT_TO_TOD_Max');

// @TEST-RUN
converted := TryConvert_LINT_TO_Destination(value, actual);
equal := actual = LINT_TO_TOD(value);

// @TEST-ASSERT
AssertTrue(Condition := equal, Message := 'Did not convert LINT to TOD correctly');
AssertTrue(Condition := converted, Message := 'Did not report LINT to TOD conversion was successful');

TEST_FINISHED();
END_METHOD

METHOD PUBLIC Check_LINT_TO_UDINT_Min
VAR
	value : LINT := DatatypeLimits.MIN_VALUE_OF_LINT_WHICH_CAN_BE_HELD_IN_A_UDINT;
	actual : UDINT;
	converted : BOOL;
	equal : BOOL;
END_VAR
TEST('Check_LINT_TO_UDINT_Min');

// @TEST-RUN
converted := TryConvert_LINT_TO_Destination(value, actual);
equal := actual = LINT_TO_UDINT(value);

// @TEST-ASSERT
AssertTrue(Condition := equal, Message := 'Did not convert LINT to UDINT correctly');
AssertTrue(Condition := converted, Message := 'Did not report LINT to UDINT conversion was successful');

TEST_FINISHED();
END_METHOD

METHOD PUBLIC Check_LINT_TO_UDINT_TooHigh
VAR
	value : LINT := DatatypeLimits.LINT_MAX_VALUE;
	actual : UDINT;
	converted : BOOL;
END_VAR
TEST('Check_LINT_TO_UDINT_TooHigh');

// @TEST-RUN
converted := TryConvert_LINT_TO_Destination(value, actual);

// @TEST-ASSERT
AssertFalse(Condition := converted, Message := 'Did not report LINT to UDINT conversion was prevented');

TEST_FINISHED();
END_METHOD

METHOD PUBLIC Check_LINT_TO_UDINT_TooLow
VAR
	value : LINT := DatatypeLimits.LINT_MIN_VALUE;
	actual : UDINT;
	converted : BOOL;
END_VAR
TEST('Check_LINT_TO_UDINT_TooLow');

// @TEST-RUN
converted := TryConvert_LINT_TO_Destination(value, actual);

// @TEST-ASSERT
AssertFalse(Condition := converted, Message := 'Did not report LINT to UDINT conversion was prevented');

TEST_FINISHED();
END_METHOD

METHOD PUBLIC Check_LINT_TO_UDINT_Max
VAR
	value : LINT := DatatypeLimits.MAX_VALUE_OF_LINT_WHICH_CAN_BE_HELD_IN_A_UDINT;
	actual : UDINT;
	converted : BOOL;
	equal : BOOL;
END_VAR
TEST('Check_LINT_TO_UDINT_Max');

// @TEST-RUN
converted := TryConvert_LINT_TO_Destination(value, actual);
equal := actual = LINT_TO_UDINT(value);

// @TEST-ASSERT
AssertTrue(Condition := equal, Message := 'Did not convert LINT to UDINT correctly');
AssertTrue(Condition := converted, Message := 'Did not report LINT to UDINT conversion was successful');

TEST_FINISHED();
END_METHOD

METHOD PUBLIC Check_LINT_TO_UINT_Min
VAR
	value : LINT := DatatypeLimits.MIN_VALUE_OF_LINT_WHICH_CAN_BE_HELD_IN_A_UINT;
	actual : UINT;
	converted : BOOL;
	equal : BOOL;
END_VAR
TEST('Check_LINT_TO_UINT_Min');

// @TEST-RUN
converted := TryConvert_LINT_TO_Destination(value, actual);
equal := actual = LINT_TO_UINT(value);

// @TEST-ASSERT
AssertTrue(Condition := equal, Message := 'Did not convert LINT to UINT correctly');
AssertTrue(Condition := converted, Message := 'Did not report LINT to UINT conversion was successful');

TEST_FINISHED();
END_METHOD

METHOD PUBLIC Check_LINT_TO_UINT_TooHigh
VAR
	value : LINT := DatatypeLimits.LINT_MAX_VALUE;
	actual : UINT;
	converted : BOOL;
END_VAR
TEST('Check_LINT_TO_UINT_TooHigh');

// @TEST-RUN
converted := TryConvert_LINT_TO_Destination(value, actual);

// @TEST-ASSERT
AssertFalse(Condition := converted, Message := 'Did not report LINT to UINT conversion was prevented');

TEST_FINISHED();
END_METHOD

METHOD PUBLIC Check_LINT_TO_UINT_TooLow
VAR
	value : LINT := DatatypeLimits.LINT_MIN_VALUE;
	actual : UINT;
	converted : BOOL;
END_VAR
TEST('Check_LINT_TO_UINT_TooLow');

// @TEST-RUN
converted := TryConvert_LINT_TO_Destination(value, actual);

// @TEST-ASSERT
AssertFalse(Condition := converted, Message := 'Did not report LINT to UINT conversion was prevented');

TEST_FINISHED();
END_METHOD

METHOD PUBLIC Check_LINT_TO_UINT_Max
VAR
	value : LINT := DatatypeLimits.MAX_VALUE_OF_LINT_WHICH_CAN_BE_HELD_IN_A_UINT;
	actual : UINT;
	converted : BOOL;
	equal : BOOL;
END_VAR
TEST('Check_LINT_TO_UINT_Max');

// @TEST-RUN
converted := TryConvert_LINT_TO_Destination(value, actual);
equal := actual = LINT_TO_UINT(value);

// @TEST-ASSERT
AssertTrue(Condition := equal, Message := 'Did not convert LINT to UINT correctly');
AssertTrue(Condition := converted, Message := 'Did not report LINT to UINT conversion was successful');

TEST_FINISHED();
END_METHOD

METHOD PUBLIC Check_LINT_TO_ULINT_Min
VAR
	value : LINT := DatatypeLimits.MIN_VALUE_OF_LINT_WHICH_CAN_BE_HELD_IN_A_ULINT;
	actual : ULINT;
	converted : BOOL;
	equal : BOOL;
END_VAR
TEST('Check_LINT_TO_ULINT_Min');

// @TEST-RUN
converted := TryConvert_LINT_TO_Destination(value, actual);
equal := actual = LINT_TO_ULINT(value);

// @TEST-ASSERT
AssertTrue(Condition := equal, Message := 'Did not convert LINT to ULINT correctly');
AssertTrue(Condition := converted, Message := 'Did not report LINT to ULINT conversion was successful');

TEST_FINISHED();
END_METHOD

METHOD PUBLIC Check_LINT_TO_ULINT_TooLow
VAR
	value : LINT := DatatypeLimits.LINT_MIN_VALUE;
	actual : ULINT;
	converted : BOOL;
END_VAR
TEST('Check_LINT_TO_ULINT_TooLow');

// @TEST-RUN
converted := TryConvert_LINT_TO_Destination(value, actual);

// @TEST-ASSERT
AssertFalse(Condition := converted, Message := 'Did not report LINT to ULINT conversion was prevented');

TEST_FINISHED();
END_METHOD

METHOD PUBLIC Check_LINT_TO_ULINT_Max
VAR
	value : LINT := DatatypeLimits.LINT_MAX_VALUE;
	actual : ULINT;
	converted : BOOL;
	equal : BOOL;
END_VAR
TEST('Check_LINT_TO_ULINT_Max');

// @TEST-RUN
converted := TryConvert_LINT_TO_Destination(value, actual);
equal := actual = LINT_TO_ULINT(value);

// @TEST-ASSERT
AssertTrue(Condition := equal, Message := 'Did not convert LINT to ULINT correctly');
AssertTrue(Condition := converted, Message := 'Did not report LINT to ULINT conversion was successful');

TEST_FINISHED();
END_METHOD

METHOD PUBLIC Check_LINT_TO_USINT_Min
VAR
	value : LINT := DatatypeLimits.MIN_VALUE_OF_LINT_WHICH_CAN_BE_HELD_IN_A_USINT;
	actual : USINT;
	converted : BOOL;
	equal : BOOL;
END_VAR
TEST('Check_LINT_TO_USINT_Min');

// @TEST-RUN
converted := TryConvert_LINT_TO_Destination(value, actual);
equal := actual = LINT_TO_USINT(value);

// @TEST-ASSERT
AssertTrue(Condition := equal, Message := 'Did not convert LINT to USINT correctly');
AssertTrue(Condition := converted, Message := 'Did not report LINT to USINT conversion was successful');

TEST_FINISHED();
END_METHOD

METHOD PUBLIC Check_LINT_TO_USINT_TooHigh
VAR
	value : LINT := DatatypeLimits.LINT_MAX_VALUE;
	actual : USINT;
	converted : BOOL;
END_VAR
TEST('Check_LINT_TO_USINT_TooHigh');

// @TEST-RUN
converted := TryConvert_LINT_TO_Destination(value, actual);

// @TEST-ASSERT
AssertFalse(Condition := converted, Message := 'Did not report LINT to USINT conversion was prevented');

TEST_FINISHED();
END_METHOD

METHOD PUBLIC Check_LINT_TO_USINT_TooLow
VAR
	value : LINT := DatatypeLimits.LINT_MIN_VALUE;
	actual : USINT;
	converted : BOOL;
END_VAR
TEST('Check_LINT_TO_USINT_TooLow');

// @TEST-RUN
converted := TryConvert_LINT_TO_Destination(value, actual);

// @TEST-ASSERT
AssertFalse(Condition := converted, Message := 'Did not report LINT to USINT conversion was prevented');

TEST_FINISHED();
END_METHOD

METHOD PUBLIC Check_LINT_TO_USINT_Max
VAR
	value : LINT := DatatypeLimits.MAX_VALUE_OF_LINT_WHICH_CAN_BE_HELD_IN_A_USINT;
	actual : USINT;
	converted : BOOL;
	equal : BOOL;
END_VAR
TEST('Check_LINT_TO_USINT_Max');

// @TEST-RUN
converted := TryConvert_LINT_TO_Destination(value, actual);
equal := actual = LINT_TO_USINT(value);

// @TEST-ASSERT
AssertTrue(Condition := equal, Message := 'Did not convert LINT to USINT correctly');
AssertTrue(Condition := converted, Message := 'Did not report LINT to USINT conversion was successful');

TEST_FINISHED();
END_METHOD

METHOD PUBLIC Check_LINT_TO_WORD_Min
VAR
	value : LINT := DatatypeLimits.MIN_VALUE_OF_LINT_WHICH_CAN_BE_HELD_IN_A_WORD;
	actual : WORD;
	converted : BOOL;
	equal : BOOL;
END_VAR
TEST('Check_LINT_TO_WORD_Min');

// @TEST-RUN
converted := TryConvert_LINT_TO_Destination(value, actual);
equal := actual = LINT_TO_WORD(value);

// @TEST-ASSERT
AssertTrue(Condition := equal, Message := 'Did not convert LINT to WORD correctly');
AssertTrue(Condition := converted, Message := 'Did not report LINT to WORD conversion was successful');

TEST_FINISHED();
END_METHOD

METHOD PUBLIC Check_LINT_TO_WORD_TooHigh
VAR
	value : LINT := DatatypeLimits.LINT_MAX_VALUE;
	actual : WORD;
	converted : BOOL;
END_VAR
TEST('Check_LINT_TO_WORD_TooHigh');

// @TEST-RUN
converted := TryConvert_LINT_TO_Destination(value, actual);

// @TEST-ASSERT
AssertFalse(Condition := converted, Message := 'Did not report LINT to WORD conversion was prevented');

TEST_FINISHED();
END_METHOD

METHOD PUBLIC Check_LINT_TO_WORD_TooLow
VAR
	value : LINT := DatatypeLimits.LINT_MIN_VALUE;
	actual : WORD;
	converted : BOOL;
END_VAR
TEST('Check_LINT_TO_WORD_TooLow');

// @TEST-RUN
converted := TryConvert_LINT_TO_Destination(value, actual);

// @TEST-ASSERT
AssertFalse(Condition := converted, Message := 'Did not report LINT to WORD conversion was prevented');

TEST_FINISHED();
END_METHOD

METHOD PUBLIC Check_LINT_TO_WORD_Max
VAR
	value : LINT := DatatypeLimits.MAX_VALUE_OF_LINT_WHICH_CAN_BE_HELD_IN_A_WORD;
	actual : WORD;
	converted : BOOL;
	equal : BOOL;
END_VAR
TEST('Check_LINT_TO_WORD_Max');

// @TEST-RUN
converted := TryConvert_LINT_TO_Destination(value, actual);
equal := actual = LINT_TO_WORD(value);

// @TEST-ASSERT
AssertTrue(Condition := equal, Message := 'Did not convert LINT to WORD correctly');
AssertTrue(Condition := converted, Message := 'Did not report LINT to WORD conversion was successful');

TEST_FINISHED();
END_METHOD

END_FUNCTION_BLOCK

// ---- Tests/USINT_TO_TestSuite.TcPOU
FUNCTION_BLOCK PUBLIC USINT_TO_TestSuite EXTENDS TcUnit.FB_TestSuite
VAR
END_VAR

Check_USINT_TO_BOOL_Max();
Check_USINT_TO_BOOL_Min();
Check_USINT_TO_BYTE_Max();
Check_USINT_TO_BYTE_Min();
Check_USINT_TO_WORD_Max();
Check_USINT_TO_WORD_Min();
Check_USINT_TO_DWORD_Max();
Check_USINT_TO_DWORD_Min();
Check_USINT_TO_LWORD_Max();
Check_USINT_TO_LWORD_Min();
Check_USINT_TO_SINT_Max();
Check_USINT_TO_SINT_Min();
Check_USINT_TO_SINT_TooHigh();
Check_USINT_TO_INT_Max();
Check_USINT_TO_INT_Min();
Check_USINT_TO_DINT_Max();
Check_USINT_TO_DINT_Min();
Check_USINT_TO_LINT_Max();
Check_USINT_TO_LINT_Min();
Check_USINT_TO_USINT_Max();
Check_USINT_TO_USINT_Min();
Check_USINT_TO_UINT_Max();
Check_USINT_TO_UINT_Min();
Check_USINT_TO_UDINT_Max();
Check_USINT_TO_UDINT_Min();
Check_USINT_TO_ULINT_Max();
Check_USINT_TO_ULINT_Min();
Check_USINT_TO_REAL_Max();
Check_USINT_TO_REAL_Min();
Check_USINT_TO_LREAL_Max();
Check_USINT_TO_LREAL_Min();
Check_USINT_TO_TIME_Max();
Check_USINT_TO_TIME_Min();
Check_USINT_TO_TOD_Max();
Check_USINT_TO_TOD_Min();
Check_USINT_TO_DATE_Max();
Check_USINT_TO_DATE_Min();
Check_USINT_TO_DT_Max();
Check_USINT_TO_DT_Min();
Check_USINT_TO_STRING_Max();
Check_USINT_TO_STRING_Min();

METHOD PUBLIC Check_USINT_TO_BOOL_Min
VAR
	value : USINT := DatatypeLimits.USINT_MIN_VALUE;
	actual : BOOL;
	converted : BOOL;
	equal : BOOL;
END_VAR
TEST('Check_USINT_TO_BOOL_Min');

// @TEST-RUN
converted := TryConvert_USINT_TO_Destination(value, actual);
equal := actual = USINT_TO_BOOL(value);

// @TEST-ASSERT
AssertTrue(Condition := equal, Message := 'Did not convert USINT to BOOL correctly');
AssertTrue(Condition := converted, Message := 'Did not report USINT to BOOL conversion was successful');

TEST_FINISHED();
END_METHOD

METHOD PUBLIC Check_USINT_TO_BOOL_Max
VAR
	value : USINT := DatatypeLimits.USINT_MAX_VALUE;
	actual : BOOL;
	converted : BOOL;
	equal : BOOL;
END_VAR
TEST('Check_USINT_TO_BOOL_Max');

// @TEST-RUN
converted := TryConvert_USINT_TO_Destination(value, actual);
equal := actual = USINT_TO_BOOL(value);

// @TEST-ASSERT
AssertTrue(Condition := equal, Message := 'Did not convert USINT to BOOL correctly');
AssertTrue(Condition := converted, Message := 'Did not report USINT to BOOL conversion was successful');

TEST_FINISHED();
END_METHOD

METHOD PUBLIC Check_USINT_TO_BYTE_Min
VAR
	value : USINT := DatatypeLimits.USINT_MIN_VALUE;
	actual : BYTE;
	converted : BOOL;
	equal : BOOL;
END_VAR
TEST('Check_USINT_TO_BYTE_Min');

// @TEST-RUN
converted := TryConvert_USINT_TO_Destination(value, actual);
equal := actual = USINT_TO_BYTE(value);

// @TEST-ASSERT
AssertTrue(Condition := equal, Message := 'Did not convert USINT to BYTE correctly');
AssertTrue(Condition := converted, Message := 'Did not report USINT to BYTE conversion was successful');

TEST_FINISHED();
END_METHOD

METHOD PUBLIC Check_USINT_TO_BYTE_Max
VAR
	value : USINT := DatatypeLimits.USINT_MAX_VALUE;
	actual : BYTE;
	converted : BOOL;
	equal : BOOL;
END_VAR
TEST('Check_USINT_TO_BYTE_Max');

// @TEST-RUN
converted := TryConvert_USINT_TO_Destination(value, actual);
equal := actual = USINT_TO_BYTE(value);

// @TEST-ASSERT
AssertTrue(Condition := equal, Message := 'Did not convert USINT to BYTE correctly');
AssertTrue(Condition := converted, Message := 'Did not report USINT to BYTE conversion was successful');

TEST_FINISHED();
END_METHOD

METHOD PUBLIC Check_USINT_TO_DATE_Min
VAR
	value : USINT := DatatypeLimits.USINT_MIN_VALUE;
	actual : DATE;
	converted : BOOL;
	equal : BOOL;
END_VAR
TEST('Check_USINT_TO_DATE_Min');

// @TEST-RUN
converted := TryConvert_USINT_TO_Destination(value, actual);
equal := actual = USINT_TO_DATE(value);

// @TEST-ASSERT
AssertTrue(Condition := equal, Message := 'Did not convert USINT to DATE correctly');
AssertTrue(Condition := converted, Message := 'Did not report USINT to DATE conversion was successful');

TEST_FINISHED();
END_METHOD

METHOD PUBLIC Check_USINT_TO_DATE_Max
VAR
	value : USINT := DatatypeLimits.USINT_MAX_VALUE;
	actual : DATE;
	converted : BOOL;
	equal : BOOL;
END_VAR
TEST('Check_USINT_TO_DATE_Max');

// @TEST-RUN
converted := TryConvert_USINT_TO_Destination(value, actual);
equal := actual = USINT_TO_DATE(value);

// @TEST-ASSERT
AssertTrue(Condition := equal, Message := 'Did not convert USINT to DATE correctly');
AssertTrue(Condition := converted, Message := 'Did not report USINT to DATE conversion was successful');

TEST_FINISHED();
END_METHOD

METHOD PUBLIC Check_USINT_TO_DINT_Min
VAR
	value : USINT := DatatypeLimits.USINT_MIN_VALUE;
	actual : DINT;
	converted : BOOL;
	equal : BOOL;
END_VAR
TEST('Check_USINT_TO_DINT_Min');

// @TEST-RUN
converted := TryConvert_USINT_TO_Destination(value, actual);
equal := actual = USINT_TO_DINT(value);

// @TEST-ASSERT
AssertTrue(Condition := equal, Message := 'Did not convert USINT to DINT correctly');
AssertTrue(Condition := converted, Message := 'Did not report USINT to DINT conversion was successful');

TEST_FINISHED();
END_METHOD

METHOD PUBLIC Check_USINT_TO_DINT_Max
VAR
	value : USINT := DatatypeLimits.USINT_MAX_VALUE;
	actual : DINT;
	converted : BOOL;
	equal : BOOL;
END_VAR
TEST('Check_USINT_TO_DINT_Max');

// @TEST-RUN
converted := TryConvert_USINT_TO_Destination(value, actual);
equal := actual = USINT_TO_DINT(value);

// @TEST-ASSERT
AssertTrue(Condition := equal, Message := 'Did not convert USINT to DINT correctly');
AssertTrue(Condition := converted, Message := 'Did not report USINT to DINT conversion was successful');

TEST_FINISHED();
END_METHOD

METHOD PUBLIC Check_USINT_TO_DT_Min
VAR
	value : USINT := DatatypeLimits.USINT_MIN_VALUE;
	actual : DT;
	converted : BOOL;
	equal : BOOL;
END_VAR
TEST('Check_USINT_TO_DT_Min');

// @TEST-RUN
converted := TryConvert_USINT_TO_Destination(value, actual);
equal := actual = USINT_TO_DT(value);

// @TEST-ASSERT
AssertTrue(Condition := equal, Message := 'Did not convert USINT to DT correctly');
AssertTrue(Condition := converted, Message := 'Did not report USINT to DT conversion was successful');

TEST_FINISHED();
END_METHOD

METHOD PUBLIC Check_USINT_TO_DT_Max
VAR
	value : USINT := DatatypeLimits.USINT_MAX_VALUE;
	actual : DT;
	converted : BOOL;
	equal : BOOL;
END_VAR
TEST('Check_USINT_TO_DT_Max');

// @TEST-RUN
converted := TryConvert_USINT_TO_Destination(value, actual);
equal := actual = USINT_TO_DT(value);

// @TEST-ASSERT
AssertTrue(Condition := equal, Message := 'Did not convert USINT to DT correctly');
AssertTrue(Condition := converted, Message := 'Did not report USINT to DT conversion was successful');

TEST_FINISHED();
END_METHOD

METHOD PUBLIC Check_USINT_TO_DWORD_Min
VAR
	value : USINT := DatatypeLimits.USINT_MIN_VALUE;
	actual : DWORD;
	converted : BOOL;
	equal : BOOL;
END_VAR
TEST('Check_USINT_TO_DWORD_Min');

// @TEST-RUN
converted := TryConvert_USINT_TO_Destination(value, actual);
equal := actual = USINT_TO_DWORD(value);

// @TEST-ASSERT
AssertTrue(Condition := equal, Message := 'Did not convert USINT to DWORD correctly');
AssertTrue(Condition := converted, Message := 'Did not report USINT to DWORD conversion was successful');

TEST_FINISHED();
END_METHOD

METHOD PUBLIC Check_USINT_TO_DWORD_Max
VAR
	value : USINT := DatatypeLimits.USINT_MAX_VALUE;
	actual : DWORD;
	converted : BOOL;
	equal : BOOL;
END_VAR
TEST('Check_USINT_TO_DWORD_Max');

// @TEST-RUN
converted := TryConvert_USINT_TO_Destination(value, actual);
equal := actual = USINT_TO_DWORD(value);

// @TEST-ASSERT
AssertTrue(Condition := equal, Message := 'Did not convert USINT to DWORD correctly');
AssertTrue(Condition := converted, Message := 'Did not report USINT to DWORD conversion was successful');

TEST_FINISHED();
END_METHOD

METHOD PUBLIC Check_USINT_TO_INT_Min
VAR
	value : USINT := DatatypeLimits.USINT_MIN_VALUE;
	actual : INT;
	converted : BOOL;
	equal : BOOL;
END_VAR
TEST('Check_USINT_TO_INT_Min');

// @TEST-RUN
converted := TryConvert_USINT_TO_Destination(value, actual);
equal := actual = USINT_TO_INT(value);

// @TEST-ASSERT
AssertTrue(Condition := equal, Message := 'Did not convert USINT to INT correctly');
AssertTrue(Condition := converted, Message := 'Did not report USINT to INT conversion was successful');

TEST_FINISHED();
END_METHOD

METHOD PUBLIC Check_USINT_TO_INT_Max
VAR
	value : USINT := DatatypeLimits.USINT_MAX_VALUE;
	actual : INT;
	converted : BOOL;
	equal : BOOL;
END_VAR
TEST('Check_USINT_TO_INT_Max');

// @TEST-RUN
converted := TryConvert_USINT_TO_Destination(value, actual);
equal := actual = USINT_TO_INT(value);

// @TEST-ASSERT
AssertTrue(Condition := equal, Message := 'Did not convert USINT to INT correctly');
AssertTrue(Condition := converted, Message := 'Did not report USINT to INT conversion was successful');

TEST_FINISHED();
END_METHOD

METHOD PUBLIC Check_USINT_TO_LINT_Min
VAR
	value : USINT := DatatypeLimits.USINT_MIN_VALUE;
	actual : LINT;
	converted : BOOL;
	equal : BOOL;
END_VAR
TEST('Check_USINT_TO_LINT_Min');

// @TEST-RUN
converted := TryConvert_USINT_TO_Destination(value, actual);
equal := actual = USINT_TO_LINT(value);

// @TEST-ASSERT
AssertTrue(Condition := equal, Message := 'Did not convert USINT to LINT correctly');
AssertTrue(Condition := converted, Message := 'Did not report USINT to LINT conversion was successful');

TEST_FINISHED();
END_METHOD

METHOD PUBLIC Check_USINT_TO_LINT_Max
VAR
	value : USINT := DatatypeLimits.USINT_MAX_VALUE;
	actual : LINT;
	converted : BOOL;
	equal : BOOL;
END_VAR
TEST('Check_USINT_TO_LINT_Max');

// @TEST-RUN
converted := TryConvert_USINT_TO_Destination(value, actual);
equal := actual = USINT_TO_LINT(value);

// @TEST-ASSERT
AssertTrue(Condition := equal, Message := 'Did not convert USINT to LINT correctly');
AssertTrue(Condition := converted, Message := 'Did not report USINT to LINT conversion was successful');

TEST_FINISHED();
END_METHOD

METHOD PUBLIC Check_USINT_TO_LREAL_Min
VAR
	value : USINT := DatatypeLimits.USINT_MIN_VALUE;
	actual : LREAL;
	converted : BOOL;
	equal : BOOL;
END_VAR
TEST('Check_USINT_TO_LREAL_Min');

// @TEST-RUN
converted := TryConvert_USINT_TO_Destination(value, actual);
equal := actual = USINT_TO_LREAL(value);

// @TEST-ASSERT
AssertTrue(Condition := equal, Message := 'Did not convert USINT to LREAL correctly');
AssertTrue(Condition := converted, Message := 'Did not report USINT to LREAL conversion was successful');

TEST_FINISHED();
END_METHOD

METHOD PUBLIC Check_USINT_TO_LREAL_Max
VAR
	value : USINT := DatatypeLimits.USINT_MAX_VALUE;
	actual : LREAL;
	converted : BOOL;
	equal : BOOL;
END_VAR
TEST('Check_USINT_TO_LREAL_Max');

// @TEST-RUN
converted := TryConvert_USINT_TO_Destination(value, actual);
equal := actual = USINT_TO_LREAL(value);

// @TEST-ASSERT
AssertTrue(Condition := equal, Message := 'Did not convert USINT to LREAL correctly');
AssertTrue(Condition := converted, Message := 'Did not report USINT to LREAL conversion was successful');

TEST_FINISHED();
END_METHOD

METHOD PUBLIC Check_USINT_TO_LWORD_Min
VAR
	value : USINT := DatatypeLimits.USINT_MIN_VALUE;
	actual : LWORD;
	converted : BOOL;
	equal : BOOL;
END_VAR
TEST('Check_USINT_TO_LWORD_Min');

// @TEST-RUN
converted := TryConvert_USINT_TO_Destination(value, actual);
equal := actual = USINT_TO_LWORD(value);

// @TEST-ASSERT
AssertTrue(Condition := equal, Message := 'Did not convert USINT to LWORD correctly');
AssertTrue(Condition := converted, Message := 'Did not report USINT to LWORD conversion was successful');

TEST_FINISHED();
END_METHOD

METHOD PUBLIC Check_USINT_TO_LWORD_Max
VAR
	value : USINT := DatatypeLimits.USINT_MAX_VALUE;
	actual : LWORD;
	converted : BOOL;
	equal : BOOL;
END_VAR
TEST('Check_USINT_TO_LWORD_Max');

// @TEST-RUN
converted := TryConvert_USINT_TO_Destination(value, actual);
equal := actual = USINT_TO_LWORD(value);

// @TEST-ASSERT
AssertTrue(Condition := equal, Message := 'Did not convert USINT to LWORD correctly');
AssertTrue(Condition := converted, Message := 'Did not report USINT to LWORD conversion was successful');

TEST_FINISHED();
END_METHOD

METHOD PUBLIC Check_USINT_TO_REAL_Min
VAR
	value : USINT := DatatypeLimits.USINT_MIN_VALUE;
	actual : REAL;
	converted : BOOL;
	equal : BOOL;
END_VAR
TEST('Check_USINT_TO_REAL_Min');

// @TEST-RUN
converted := TryConvert_USINT_TO_Destination(value, actual);
equal := actual = USINT_TO_REAL(value);

// @TEST-ASSERT
AssertTrue(Condition := equal, Message := 'Did not convert USINT to REAL correctly');
AssertTrue(Condition := converted, Message := 'Did not report USINT to REAL conversion was successful');

TEST_FINISHED();
END_METHOD

METHOD PUBLIC Check_USINT_TO_REAL_Max
VAR
	value : USINT := DatatypeLimits.USINT_MAX_VALUE;
	actual : REAL;
	converted : BOOL;
	equal : BOOL;
END_VAR
TEST('Check_USINT_TO_REAL_Max');

// @TEST-RUN
converted := TryConvert_USINT_TO_Destination(value, actual);
equal := actual = USINT_TO_REAL(value);

// @TEST-ASSERT
AssertTrue(Condition := equal, Message := 'Did not convert USINT to REAL correctly');
AssertTrue(Condition := converted, Message := 'Did not report USINT to REAL conversion was successful');

TEST_FINISHED();
END_METHOD

METHOD PUBLIC Check_USINT_TO_SINT_Min
VAR
	value : USINT := DatatypeLimits.USINT_MIN_VALUE;
	actual : SINT;
	converted : BOOL;
	equal : BOOL;
END_VAR
TEST('Check_USINT_TO_SINT_Min');

// @TEST-RUN
converted := TryConvert_USINT_TO_Destination(value, actual);
equal := actual = USINT_TO_SINT(value);

// @TEST-ASSERT
AssertTrue(Condition := equal, Message := 'Did not convert USINT to SINT correctly');
AssertTrue(Condition := converted, Message := 'Did not report USINT to SINT conversion was successful');

TEST_FINISHED();
END_METHOD

METHOD PUBLIC Check_USINT_TO_SINT_TooHigh
VAR
	value : USINT := DatatypeLimits.USINT_MAX_VALUE;
	actual : SINT;
	converted : BOOL;
END_VAR
TEST('Check_USINT_TO_SINT_TooHigh');

// @TEST-RUN
converted := TryConvert_USINT_TO_Destination(value, actual);

// @TEST-ASSERT
AssertFalse(Condition := converted, Message := 'Did not report USINT to SINT conversion was prevented');

TEST_FINISHED();
END_METHOD

METHOD PUBLIC Check_USINT_TO_SINT_Max
VAR
	value : USINT := DatatypeLimits.MAX_VALUE_OF_USINT_WHICH_CAN_BE_HELD_IN_A_SINT;
	actual : SINT;
	converted : BOOL;
	equal : BOOL;
END_VAR
TEST('Check_USINT_TO_SINT_Max');

// @TEST-RUN
converted := TryConvert_USINT_TO_Destination(value, actual);
equal := actual = USINT_TO_SINT(value);

// @TEST-ASSERT
AssertTrue(Condition := equal, Message := 'Did not convert USINT to SINT correctly');
AssertTrue(Condition := converted, Message := 'Did not report USINT to SINT conversion was successful');

TEST_FINISHED();
END_METHOD

METHOD PUBLIC Check_USINT_TO_STRING_Min
VAR
	value : USINT := DatatypeLimits.USINT_MIN_VALUE;
	actual : STRING;
	converted : BOOL;
	equal : BOOL;
END_VAR
TEST('Check_USINT_TO_STRING_Min');

// @TEST-RUN
converted := TryConvert_USINT_TO_Destination(value, actual);
equal := actual = USINT_TO_STRING(value);

// @TEST-ASSERT
AssertTrue(Condition := equal, Message := 'Did not convert USINT to STRING correctly');
AssertTrue(Condition := converted, Message := 'Did not report USINT to STRING conversion was successful');

TEST_FINISHED();
END_METHOD

METHOD PUBLIC Check_USINT_TO_STRING_Max
VAR
	value : USINT := DatatypeLimits.USINT_MAX_VALUE;
	actual : STRING;
	converted : BOOL;
	equal : BOOL;
END_VAR
TEST('Check_USINT_TO_STRING_Max');

// @TEST-RUN
converted := TryConvert_USINT_TO_Destination(value, actual);
equal := actual = USINT_TO_STRING(value);

// @TEST-ASSERT
AssertTrue(Condition := equal, Message := 'Did not convert USINT to STRING correctly');
AssertTrue(Condition := converted, Message := 'Did not report USINT to STRING conversion was successful');

TEST_FINISHED();
END_METHOD

METHOD PUBLIC Check_USINT_TO_TIME_Min
VAR
	value : USINT := DatatypeLimits.USINT_MIN_VALUE;
	actual : TIME;
	converted : BOOL;
	equal : BOOL;
END_VAR
TEST('Check_USINT_TO_TIME_Min');

// @TEST-RUN
converted := TryConvert_USINT_TO_Destination(value, actual);
equal := actual = USINT_TO_TIME(value);

// @TEST-ASSERT
AssertTrue(Condition := equal, Message := 'Did not convert USINT to TIME correctly');
AssertTrue(Condition := converted, Message := 'Did not report USINT to TIME conversion was successful');

TEST_FINISHED();
END_METHOD

METHOD PUBLIC Check_USINT_TO_TIME_Max
VAR
	value : USINT := DatatypeLimits.USINT_MAX_VALUE;
	actual : TIME;
	converted : BOOL;
	equal : BOOL;
END_VAR
TEST('Check_USINT_TO_TIME_Max');

// @TEST-RUN
converted := TryConvert_USINT_TO_Destination(value, actual);
equal := actual = USINT_TO_TIME(value);

// @TEST-ASSERT
AssertTrue(Condition := equal, Message := 'Did not convert USINT to TIME correctly');
AssertTrue(Condition := converted, Message := 'Did not report USINT to TIME conversion was successful');

TEST_FINISHED();
END_METHOD

METHOD PUBLIC Check_USINT_TO_TOD_Min
VAR
	value : USINT := DatatypeLimits.USINT_MIN_VALUE;
	actual : TOD;
	converted : BOOL;
	equal : BOOL;
END_VAR
TEST('Check_USINT_TO_TOD_Min');

// @TEST-RUN
converted := TryConvert_USINT_TO_Destination(value, actual);
equal := actual = USINT_TO_TOD(value);

// @TEST-ASSERT
AssertTrue(Condition := equal, Message := 'Did not convert USINT to TOD correctly');
AssertTrue(Condition := converted, Message := 'Did not report USINT to TOD conversion was successful');

TEST_FINISHED();
END_METHOD

METHOD PUBLIC Check_USINT_TO_TOD_Max
VAR
	value : USINT := DatatypeLimits.USINT_MAX_VALUE;
	actual : TOD;
	converted : BOOL;
	equal : BOOL;
END_VAR
TEST('Check_USINT_TO_TOD_Max');

// @TEST-RUN
converted := TryConvert_USINT_TO_Destination(value, actual);
equal := actual = USINT_TO_TOD(value);

// @TEST-ASSERT
AssertTrue(Condition := equal, Message := 'Did not convert USINT to TOD correctly');
AssertTrue(Condition := converted, Message := 'Did not report USINT to TOD conversion was successful');

TEST_FINISHED();
END_METHOD

METHOD PUBLIC Check_USINT_TO_UDINT_Min
VAR
	value : USINT := DatatypeLimits.USINT_MIN_VALUE;
	actual : UDINT;
	converted : BOOL;
	equal : BOOL;
END_VAR
TEST('Check_USINT_TO_UDINT_Min');

// @TEST-RUN
converted := TryConvert_USINT_TO_Destination(value, actual);
equal := actual = USINT_TO_UDINT(value);

// @TEST-ASSERT
AssertTrue(Condition := equal, Message := 'Did not convert USINT to UDINT correctly');
AssertTrue(Condition := converted, Message := 'Did not report USINT to UDINT conversion was successful');

TEST_FINISHED();
END_METHOD

METHOD PUBLIC Check_USINT_TO_UDINT_Max
VAR
	value : USINT := DatatypeLimits.USINT_MAX_VALUE;
	actual : UDINT;
	converted : BOOL;
	equal : BOOL;
END_VAR
TEST('Check_USINT_TO_UDINT_Max');

// @TEST-RUN
converted := TryConvert_USINT_TO_Destination(value, actual);
equal := actual = USINT_TO_UDINT(value);

// @TEST-ASSERT
AssertTrue(Condition := equal, Message := 'Did not convert USINT to UDINT correctly');
AssertTrue(Condition := converted, Message := 'Did not report USINT to UDINT conversion was successful');

TEST_FINISHED();
END_METHOD

METHOD PUBLIC Check_USINT_TO_UINT_Min
VAR
	value : USINT := DatatypeLimits.USINT_MIN_VALUE;
	actual : UINT;
	converted : BOOL;
	equal : BOOL;
END_VAR
TEST('Check_USINT_TO_UINT_Min');

// @TEST-RUN
converted := TryConvert_USINT_TO_Destination(value, actual);
equal := actual = USINT_TO_UINT(value);

// @TEST-ASSERT
AssertTrue(Condition := equal, Message := 'Did not convert USINT to UINT correctly');
AssertTrue(Condition := converted, Message := 'Did not report USINT to UINT conversion was successful');

TEST_FINISHED();
END_METHOD

METHOD PUBLIC Check_USINT_TO_UINT_Max
VAR
	value : USINT := DatatypeLimits.USINT_MAX_VALUE;
	actual : UINT;
	converted : BOOL;
	equal : BOOL;
END_VAR
TEST('Check_USINT_TO_UINT_Max');

// @TEST-RUN
converted := TryConvert_USINT_TO_Destination(value, actual);
equal := actual = USINT_TO_UINT(value);

// @TEST-ASSERT
AssertTrue(Condition := equal, Message := 'Did not convert USINT to UINT correctly');
AssertTrue(Condition := converted, Message := 'Did not report USINT to UINT conversion was successful');

TEST_FINISHED();
END_METHOD

METHOD PUBLIC Check_USINT_TO_ULINT_Min
VAR
	value : USINT := DatatypeLimits.USINT_MIN_VALUE;
	actual : ULINT;
	converted : BOOL;
	equal : BOOL;
END_VAR
TEST('Check_USINT_TO_ULINT_Min');

// @TEST-RUN
converted := TryConvert_USINT_TO_Destination(value, actual);
equal := actual = USINT_TO_ULINT(value);

// @TEST-ASSERT
AssertTrue(Condition := equal, Message := 'Did not convert USINT to ULINT correctly');
AssertTrue(Condition := converted, Message := 'Did not report USINT to ULINT conversion was successful');

TEST_FINISHED();
END_METHOD

METHOD PUBLIC Check_USINT_TO_ULINT_Max
VAR
	value : USINT := DatatypeLimits.USINT_MAX_VALUE;
	actual : ULINT;
	converted : BOOL;
	equal : BOOL;
END_VAR
TEST('Check_USINT_TO_ULINT_Max');

// @TEST-RUN
converted := TryConvert_USINT_TO_Destination(value, actual);
equal := actual = USINT_TO_ULINT(value);

// @TEST-ASSERT
AssertTrue(Condition := equal, Message := 'Did not convert USINT to ULINT correctly');
AssertTrue(Condition := converted, Message := 'Did not report USINT to ULINT conversion was successful');

TEST_FINISHED();
END_METHOD

METHOD PUBLIC Check_USINT_TO_USINT_Min
VAR
	value : USINT := DatatypeLimits.USINT_MIN_VALUE;
	actual : USINT;
	converted : BOOL;
	equal : BOOL;
END_VAR
TEST('Check_USINT_TO_USINT_Min');

// @TEST-RUN
converted := TryConvert_USINT_TO_Destination(value, actual);
equal := actual = value;

// @TEST-ASSERT
AssertTrue(Condition := equal, Message := 'Did not convert USINT to USINT correctly');
AssertTrue(Condition := converted, Message := 'Did not report USINT to USINT conversion was successful');

TEST_FINISHED();
END_METHOD

METHOD PUBLIC Check_USINT_TO_USINT_Max
VAR
	value : USINT := DatatypeLimits.USINT_MAX_VALUE;
	actual : USINT;
	converted : BOOL;
	equal : BOOL;
END_VAR
TEST('Check_USINT_TO_USINT_Max');

// @TEST-RUN
converted := TryConvert_USINT_TO_Destination(value, actual);
equal := actual = value;

// @TEST-ASSERT
AssertTrue(Condition := equal, Message := 'Did not convert USINT to USINT correctly');
AssertTrue(Condition := converted, Message := 'Did not report USINT to USINT conversion was successful');

TEST_FINISHED();
END_METHOD

METHOD PUBLIC Check_USINT_TO_WORD_Min
VAR
	value : USINT := DatatypeLimits.USINT_MIN_VALUE;
	actual : WORD;
	converted : BOOL;
	equal : BOOL;
END_VAR
TEST('Check_USINT_TO_WORD_Min');

// @TEST-RUN
converted := TryConvert_USINT_TO_Destination(value, actual);
equal := actual = USINT_TO_WORD(value);

// @TEST-ASSERT
AssertTrue(Condition := equal, Message := 'Did not convert USINT to WORD correctly');
AssertTrue(Condition := converted, Message := 'Did not report USINT to WORD conversion was successful');

TEST_FINISHED();
END_METHOD

METHOD PUBLIC Check_USINT_TO_WORD_Max
VAR
	value : USINT := DatatypeLimits.USINT_MAX_VALUE;
	actual : WORD;
	converted : BOOL;
	equal : BOOL;
END_VAR
TEST('Check_USINT_TO_WORD_Max');

// @TEST-RUN
converted := TryConvert_USINT_TO_Destination(value, actual);
equal := actual = USINT_TO_WORD(value);

// @TEST-ASSERT
AssertTrue(Condition := equal, Message := 'Did not convert USINT to WORD correctly');
AssertTrue(Condition := converted, Message := 'Did not report USINT to WORD conversion was successful');

TEST_FINISHED();
END_METHOD

END_FUNCTION_BLOCK

// ---- Tests/UINT_TO_TestSuite.TcPOU
FUNCTION_BLOCK PUBLIC UINT_TO_TestSuite EXTENDS TcUnit.FB_TestSuite
VAR
END_VAR

Check_UINT_TO_BOOL_Max();
Check_UINT_TO_BOOL_Min();
Check_UINT_TO_BYTE_Max();
Check_UINT_TO_BYTE_Min();
Check_UINT_TO_BYTE_TooHigh();
Check_UINT_TO_WORD_Max();
Check_UINT_TO_WORD_Min();
Check_UINT_TO_DWORD_Max();
Check_UINT_TO_DWORD_Min();
Check_UINT_TO_LWORD_Max();
Check_UINT_TO_LWORD_Min();
Check_UINT_TO_SINT_Max();
Check_UINT_TO_SINT_Min();
Check_UINT_TO_SINT_TooHigh();
Check_UINT_TO_INT_Max();
Check_UINT_TO_INT_Min();
Check_UINT_TO_INT_TooHigh();
Check_UINT_TO_DINT_Max();
Check_UINT_TO_DINT_Min();
Check_UINT_TO_LINT_Max();
Check_UINT_TO_LINT_Min();
Check_UINT_TO_USINT_Max();
Check_UINT_TO_USINT_Min();
Check_UINT_TO_USINT_TooHigh();
Check_UINT_TO_UINT_Max();
Check_UINT_TO_UINT_Min();
Check_UINT_TO_UDINT_Max();
Check_UINT_TO_UDINT_Min();
Check_UINT_TO_ULINT_Max();
Check_UINT_TO_ULINT_Min();
Check_UINT_TO_REAL_Max();
Check_UINT_TO_REAL_Min();
Check_UINT_TO_LREAL_Max();
Check_UINT_TO_LREAL_Min();
Check_UINT_TO_TIME_Max();
Check_UINT_TO_TIME_Min();
Check_UINT_TO_TOD_Max();
Check_UINT_TO_TOD_Min();
Check_UINT_TO_DATE_Max();
Check_UINT_TO_DATE_Min();
Check_UINT_TO_DT_Max();
Check_UINT_TO_DT_Min();
Check_UINT_TO_STRING_Max();
Check_UINT_TO_STRING_Min();

METHOD PUBLIC Check_UINT_TO_BOOL_Min
VAR
	value : UINT := DatatypeLimits.UINT_MIN_VALUE;
	actual : BOOL;
	converted : BOOL;
	equal : BOOL;
END_VAR
TEST('Check_UINT_TO_BOOL_Min');

// @TEST-RUN
converted := TryConvert_UINT_TO_Destination(value, actual);
equal := actual = UINT_TO_BOOL(value);

// @TEST-ASSERT
AssertTrue(Condition := equal, Message := 'Did not convert UINT to BOOL correctly');
AssertTrue(Condition := converted, Message := 'Did not report UINT to BOOL conversion was successful');

TEST_FINISHED();
END_METHOD

METHOD PUBLIC Check_UINT_TO_BOOL_Max
VAR
	value : UINT := DatatypeLimits.UINT_MAX_VALUE;
	actual : BOOL;
	converted : BOOL;
	equal : BOOL;
END_VAR
TEST('Check_UINT_TO_BOOL_Max');

// @TEST-RUN
converted := TryConvert_UINT_TO_Destination(value, actual);
equal := actual = UINT_TO_BOOL(value);

// @TEST-ASSERT
AssertTrue(Condition := equal, Message := 'Did not convert UINT to BOOL correctly');
AssertTrue(Condition := converted, Message := 'Did not report UINT to BOOL conversion was successful');

TEST_FINISHED();
END_METHOD

METHOD PUBLIC Check_UINT_TO_BYTE_Min
VAR
	value : UINT := DatatypeLimits.UINT_MIN_VALUE;
	actual : BYTE;
	converted : BOOL;
	equal : BOOL;
END_VAR
TEST('Check_UINT_TO_BYTE_Min');

// @TEST-RUN
converted := TryConvert_UINT_TO_Destination(value, actual);
equal := actual = UINT_TO_BYTE(value);

// @TEST-ASSERT
AssertTrue(Condition := equal, Message := 'Did not convert UINT to BYTE correctly');
AssertTrue(Condition := converted, Message := 'Did not report UINT to BYTE conversion was successful');

TEST_FINISHED();
END_METHOD

METHOD PUBLIC Check_UINT_TO_BYTE_TooHigh
VAR
	value : UINT := DatatypeLimits.UINT_MAX_VALUE;
	actual : BYTE;
	converted : BOOL;
END_VAR
TEST('Check_UINT_TO_BYTE_TooHigh');

// @TEST-RUN
converted := TryConvert_UINT_TO_Destination(value, actual);

// @TEST-ASSERT
AssertFalse(Condition := converted, Message := 'Did not report UINT to BYTE conversion was prevented');

TEST_FINISHED();
END_METHOD

METHOD PUBLIC Check_UINT_TO_BYTE_Max
VAR
	value : UINT := DatatypeLimits.MAX_VALUE_OF_UINT_WHICH_CAN_BE_HELD_IN_A_BYTE;
	actual : BYTE;
	converted : BOOL;
	equal : BOOL;
END_VAR
TEST('Check_UINT_TO_BYTE_Max');

// @TEST-RUN
converted := TryConvert_UINT_TO_Destination(value, actual);
equal := actual = UINT_TO_BYTE(value);

// @TEST-ASSERT
AssertTrue(Condition := equal, Message := 'Did not convert UINT to BYTE correctly');
AssertTrue(Condition := converted, Message := 'Did not report UINT to BYTE conversion was successful');

TEST_FINISHED();
END_METHOD

METHOD PUBLIC Check_UINT_TO_DATE_Min
VAR
	value : UINT := DatatypeLimits.UINT_MIN_VALUE;
	actual : DATE;
	converted : BOOL;
	equal : BOOL;
END_VAR
TEST('Check_UINT_TO_DATE_Min');

// @TEST-RUN
converted := TryConvert_UINT_TO_Destination(value, actual);
equal := actual = UINT_TO_DATE(value);

// @TEST-ASSERT
AssertTrue(Condition := equal, Message := 'Did not convert UINT to DATE correctly');
AssertTrue(Condition := converted, Message := 'Did not report UINT to DATE conversion was successful');

TEST_FINISHED();
END_METHOD

METHOD PUBLIC Check_UINT_TO_DATE_Max
VAR
	value : UINT := DatatypeLimits.UINT_MAX_VALUE;
	actual : DATE;
	converted : BOOL;
	equal : BOOL;
END_VAR
TEST('Check_UINT_TO_DATE_Max');

// @TEST-RUN
converted := TryConvert_UINT_TO_Destination(value, actual);
equal := actual = UINT_TO_DATE(value);

// @TEST-ASSERT
AssertTrue(Condition := equal, Message := 'Did not convert UINT to DATE correctly');
AssertTrue(Condition := converted, Message := 'Did not report UINT to DATE conversion was successful');

TEST_FINISHED();
END_METHOD

METHOD PUBLIC Check_UINT_TO_DINT_Min
VAR
	value : UINT := DatatypeLimits.UINT_MIN_VALUE;
	actual : DINT;
	converted : BOOL;
	equal : BOOL;
END_VAR
TEST('Check_UINT_TO_DINT_Min');

// @TEST-RUN
converted := TryConvert_UINT_TO_Destination(value, actual);
equal := actual = UINT_TO_DINT(value);

// @TEST-ASSERT
AssertTrue(Condition := equal, Message := 'Did not convert UINT to DINT correctly');
AssertTrue(Condition := converted, Message := 'Did not report UINT to DINT conversion was successful');

TEST_FINISHED();
END_METHOD

METHOD PUBLIC Check_UINT_TO_DINT_Max
VAR
	value : UINT := DatatypeLimits.UINT_MAX_VALUE;
	actual : DINT;
	converted : BOOL;
	equal : BOOL;
END_VAR
TEST('Check_UINT_TO_DINT_Max');

// @TEST-RUN
converted := TryConvert_UINT_TO_Destination(value, actual);
equal := actual = UINT_TO_DINT(value);

// @TEST-ASSERT
AssertTrue(Condition := equal, Message := 'Did not convert UINT to DINT correctly');
AssertTrue(Condition := converted, Message := 'Did not report UINT to DINT conversion was successful');

TEST_FINISHED();
END_METHOD

METHOD PUBLIC Check_UINT_TO_DT_Min
VAR
	value : UINT := DatatypeLimits.UINT_MIN_VALUE;
	actual : DT;
	converted : BOOL;
	equal : BOOL;
END_VAR
TEST('Check_UINT_TO_DT_Min');

// @TEST-RUN
converted := TryConvert_UINT_TO_Destination(value, actual);
equal := actual = UINT_TO_DT(value);

// @TEST-ASSERT
AssertTrue(Condition := equal, Message := 'Did not convert UINT to DT correctly');
AssertTrue(Condition := converted, Message := 'Did not report UINT to DT conversion was successful');

TEST_FINISHED();
END_METHOD

METHOD PUBLIC Check_UINT_TO_DT_Max
VAR
	value : UINT := DatatypeLimits.UINT_MAX_VALUE;
	actual : DT;
	converted : BOOL;
	equal : BOOL;
END_VAR
TEST('Check_UINT_TO_DT_Max');

// @TEST-RUN
converted := TryConvert_UINT_TO_Destination(value, actual);
equal := actual = UINT_TO_DT(value);

// @TEST-ASSERT
AssertTrue(Condition := equal, Message := 'Did not convert UINT to DT correctly');
AssertTrue(Condition := converted, Message := 'Did not report UINT to DT conversion was successful');

TEST_FINISHED();
END_METHOD

METHOD PUBLIC Check_UINT_TO_DWORD_Min
VAR
	value : UINT := DatatypeLimits.UINT_MIN_VALUE;
	actual : DWORD;
	converted : BOOL;
	equal : BOOL;
END_VAR
TEST('Check_UINT_TO_DWORD_Min');

// @TEST-RUN
converted := TryConvert_UINT_TO_Destination(value, actual);
equal := actual = UINT_TO_DWORD(value);

// @TEST-ASSERT
AssertTrue(Condition := equal, Message := 'Did not convert UINT to DWORD correctly');
AssertTrue(Condition := converted, Message := 'Did not report UINT to DWORD conversion was successful');

TEST_FINISHED();
END_METHOD

METHOD PUBLIC Check_UINT_TO_DWORD_Max
VAR
	value : UINT := DatatypeLimits.UINT_MAX_VALUE;
	actual : DWORD;
	converted : BOOL;
	equal : BOOL;
END_VAR
TEST('Check_UINT_TO_DWORD_Max');

// @TEST-RUN
converted := TryConvert_UINT_TO_Destination(value, actual);
equal := actual = UINT_TO_DWORD(value);

// @TEST-ASSERT
AssertTrue(Condition := equal, Message := 'Did not convert UINT to DWORD correctly');
AssertTrue(Condition := converted, Message := 'Did not report UINT to DWORD conversion was successful');

TEST_FINISHED();
END_METHOD

METHOD PUBLIC Check_UINT_TO_INT_Min
VAR
	value : UINT := DatatypeLimits.UINT_MIN_VALUE;
	actual : INT;
	converted : BOOL;
	equal : BOOL;
END_VAR
TEST('Check_UINT_TO_INT_Min');

// @TEST-RUN
converted := TryConvert_UINT_TO_Destination(value, actual);
equal := actual = UINT_TO_INT(value);

// @TEST-ASSERT
AssertTrue(Condition := equal, Message := 'Did not convert UINT to INT correctly');
AssertTrue(Condition := converted, Message := 'Did not report UINT to INT conversion was successful');

TEST_FINISHED();
END_METHOD

METHOD PUBLIC Check_UINT_TO_INT_TooHigh
VAR
	value : UINT := DatatypeLimits.UINT_MAX_VALUE;
	actual : INT;
	converted : BOOL;
END_VAR
TEST('Check_UINT_TO_INT_TooHigh');

// @TEST-RUN
converted := TryConvert_UINT_TO_Destination(value, actual);

// @TEST-ASSERT
AssertFalse(Condition := converted, Message := 'Did not report UINT to INT conversion was prevented');

TEST_FINISHED();
END_METHOD

METHOD PUBLIC Check_UINT_TO_INT_Max
VAR
	value : UINT := DatatypeLimits.MAX_VALUE_OF_UINT_WHICH_CAN_BE_HELD_IN_A_INT;
	actual : INT;
	converted : BOOL;
	equal : BOOL;
END_VAR
TEST('Check_UINT_TO_INT_Max');

// @TEST-RUN
converted := TryConvert_UINT_TO_Destination(value, actual);
equal := actual = UINT_TO_INT(value);

// @TEST-ASSERT
AssertTrue(Condition := equal, Message := 'Did not convert UINT to INT correctly');
AssertTrue(Condition := converted, Message := 'Did not report UINT to INT conversion was successful');

TEST_FINISHED();
END_METHOD

METHOD PUBLIC Check_UINT_TO_LINT_Min
VAR
	value : UINT := DatatypeLimits.UINT_MIN_VALUE;
	actual : LINT;
	converted : BOOL;
	equal : BOOL;
END_VAR
TEST('Check_UINT_TO_LINT_Min');

// @TEST-RUN
converted := TryConvert_UINT_TO_Destination(value, actual);
equal := actual = UINT_TO_LINT(value);

// @TEST-ASSERT
AssertTrue(Condition := equal, Message := 'Did not convert UINT to LINT correctly');
AssertTrue(Condition := converted, Message := 'Did not report UINT to LINT conversion was successful');

TEST_FINISHED();
END_METHOD

METHOD PUBLIC Check_UINT_TO_LINT_Max
VAR
	value : UINT := DatatypeLimits.UINT_MAX_VALUE;
	actual : LINT;
	converted : BOOL;
	equal : BOOL;
END_VAR
TEST('Check_UINT_TO_LINT_Max');

// @TEST-RUN
converted := TryConvert_UINT_TO_Destination(value, actual);
equal := actual = UINT_TO_LINT(value);

// @TEST-ASSERT
AssertTrue(Condition := equal, Message := 'Did not convert UINT to LINT correctly');
AssertTrue(Condition := converted, Message := 'Did not report UINT to LINT conversion was successful');

TEST_FINISHED();
END_METHOD

METHOD PUBLIC Check_UINT_TO_LREAL_Min
VAR
	value : UINT := DatatypeLimits.UINT_MIN_VALUE;
	actual : LREAL;
	converted : BOOL;
	equal : BOOL;
END_VAR
TEST('Check_UINT_TO_LREAL_Min');

// @TEST-RUN
converted := TryConvert_UINT_TO_Destination(value, actual);
equal := actual = UINT_TO_LREAL(value);

// @TEST-ASSERT
AssertTrue(Condition := equal, Message := 'Did not convert UINT to LREAL correctly');
AssertTrue(Condition := converted, Message := 'Did not report UINT to LREAL conversion was successful');

TEST_FINISHED();
END_METHOD

METHOD PUBLIC Check_UINT_TO_LREAL_Max
VAR
	value : UINT := DatatypeLimits.UINT_MAX_VALUE;
	actual : LREAL;
	converted : BOOL;
	equal : BOOL;
END_VAR
TEST('Check_UINT_TO_LREAL_Max');

// @TEST-RUN
converted := TryConvert_UINT_TO_Destination(value, actual);
equal := actual = UINT_TO_LREAL(value);

// @TEST-ASSERT
AssertTrue(Condition := equal, Message := 'Did not convert UINT to LREAL correctly');
AssertTrue(Condition := converted, Message := 'Did not report UINT to LREAL conversion was successful');

TEST_FINISHED();
END_METHOD

METHOD PUBLIC Check_UINT_TO_LWORD_Min
VAR
	value : UINT := DatatypeLimits.UINT_MIN_VALUE;
	actual : LWORD;
	converted : BOOL;
	equal : BOOL;
END_VAR
TEST('Check_UINT_TO_LWORD_Min');

// @TEST-RUN
converted := TryConvert_UINT_TO_Destination(value, actual);
equal := actual = UINT_TO_LWORD(value);

// @TEST-ASSERT
AssertTrue(Condition := equal, Message := 'Did not convert UINT to LWORD correctly');
AssertTrue(Condition := converted, Message := 'Did not report UINT to LWORD conversion was successful');

TEST_FINISHED();
END_METHOD

METHOD PUBLIC Check_UINT_TO_LWORD_Max
VAR
	value : UINT := DatatypeLimits.UINT_MAX_VALUE;
	actual : LWORD;
	converted : BOOL;
	equal : BOOL;
END_VAR
TEST('Check_UINT_TO_LWORD_Max');

// @TEST-RUN
converted := TryConvert_UINT_TO_Destination(value, actual);
equal := actual = UINT_TO_LWORD(value);

// @TEST-ASSERT
AssertTrue(Condition := equal, Message := 'Did not convert UINT to LWORD correctly');
AssertTrue(Condition := converted, Message := 'Did not report UINT to LWORD conversion was successful');

TEST_FINISHED();
END_METHOD

METHOD PUBLIC Check_UINT_TO_REAL_Min
VAR
	value : UINT := DatatypeLimits.UINT_MIN_VALUE;
	actual : REAL;
	converted : BOOL;
	equal : BOOL;
END_VAR
TEST('Check_UINT_TO_REAL_Min');

// @TEST-RUN
converted := TryConvert_UINT_TO_Destination(value, actual);
equal := actual = UINT_TO_REAL(value);

// @TEST-ASSERT
AssertTrue(Condition := equal, Message := 'Did not convert UINT to REAL correctly');
AssertTrue(Condition := converted, Message := 'Did not report UINT to REAL conversion was successful');

TEST_FINISHED();
END_METHOD

METHOD PUBLIC Check_UINT_TO_REAL_Max
VAR
	value : UINT := DatatypeLimits.UINT_MAX_VALUE;
	actual : REAL;
	converted : BOOL;
	equal : BOOL;
END_VAR
TEST('Check_UINT_TO_REAL_Max');

// @TEST-RUN
converted := TryConvert_UINT_TO_Destination(value, actual);
equal := actual = UINT_TO_REAL(value);

// @TEST-ASSERT
AssertTrue(Condition := equal, Message := 'Did not convert UINT to REAL correctly');
AssertTrue(Condition := converted, Message := 'Did not report UINT to REAL conversion was successful');

TEST_FINISHED();
END_METHOD

METHOD PUBLIC Check_UINT_TO_SINT_Min
VAR
	value : UINT := DatatypeLimits.UINT_MIN_VALUE;
	actual : SINT;
	converted : BOOL;
	equal : BOOL;
END_VAR
TEST('Check_UINT_TO_SINT_Min');

// @TEST-RUN
converted := TryConvert_UINT_TO_Destination(value, actual);
equal := actual = UINT_TO_SINT(value);

// @TEST-ASSERT
AssertTrue(Condition := equal, Message := 'Did not convert UINT to SINT correctly');
AssertTrue(Condition := converted, Message := 'Did not report UINT to SINT conversion was successful');

TEST_FINISHED();
END_METHOD

METHOD PUBLIC Check_UINT_TO_SINT_TooHigh
VAR
	value : UINT := DatatypeLimits.UINT_MAX_VALUE;
	actual : SINT;
	converted : BOOL;
END_VAR
TEST('Check_UINT_TO_SINT_TooHigh');

// @TEST-RUN
converted := TryConvert_UINT_TO_Destination(value, actual);

// @TEST-ASSERT
AssertFalse(Condition := converted, Message := 'Did not report UINT to SINT conversion was prevented');

TEST_FINISHED();
END_METHOD

METHOD PUBLIC Check_UINT_TO_SINT_Max
VAR
	value : UINT := DatatypeLimits.MAX_VALUE_OF_UINT_WHICH_CAN_BE_HELD_IN_A_SINT;
	actual : SINT;
	converted : BOOL;
	equal : BOOL;
END_VAR
TEST('Check_UINT_TO_SINT_Max');

// @TEST-RUN
converted := TryConvert_UINT_TO_Destination(value, actual);
equal := actual = UINT_TO_SINT(value);

// @TEST-ASSERT
AssertTrue(Condition := equal, Message := 'Did not convert UINT to SINT correctly');
AssertTrue(Condition := converted, Message := 'Did not report UINT to SINT conversion was successful');

TEST_FINISHED();
END_METHOD

METHOD PUBLIC Check_UINT_TO_STRING_Min
VAR
	value : UINT := DatatypeLimits.UINT_MIN_VALUE;
	actual : STRING;
	converted : BOOL;
	equal : BOOL;
END_VAR
TEST('Check_UINT_TO_STRING_Min');

// @TEST-RUN
converted := TryConvert_UINT_TO_Destination(value, actual);
equal := actual = UINT_TO_STRING(value);

// @TEST-ASSERT
AssertTrue(Condition := equal, Message := 'Did not convert UINT to STRING correctly');
AssertTrue(Condition := converted, Message := 'Did not report UINT to STRING conversion was successful');

TEST_FINISHED();
END_METHOD

METHOD PUBLIC Check_UINT_TO_STRING_Max
VAR
	value : UINT := DatatypeLimits.UINT_MAX_VALUE;
	actual : STRING;
	converted : BOOL;
	equal : BOOL;
END_VAR
TEST('Check_UINT_TO_STRING_Max');

// @TEST-RUN
converted := TryConvert_UINT_TO_Destination(value, actual);
equal := actual = UINT_TO_STRING(value);

// @TEST-ASSERT
AssertTrue(Condition := equal, Message := 'Did not convert UINT to STRING correctly');
AssertTrue(Condition := converted, Message := 'Did not report UINT to STRING conversion was successful');

TEST_FINISHED();
END_METHOD

METHOD PUBLIC Check_UINT_TO_TIME_Min
VAR
	value : UINT := DatatypeLimits.UINT_MIN_VALUE;
	actual : TIME;
	converted : BOOL;
	equal : BOOL;
END_VAR
TEST('Check_UINT_TO_TIME_Min');

// @TEST-RUN
converted := TryConvert_UINT_TO_Destination(value, actual);
equal := actual = UINT_TO_TIME(value);

// @TEST-ASSERT
AssertTrue(Condition := equal, Message := 'Did not convert UINT to TIME correctly');
AssertTrue(Condition := converted, Message := 'Did not report UINT to TIME conversion was successful');

TEST_FINISHED();
END_METHOD

METHOD PUBLIC Check_UINT_TO_TIME_Max
VAR
	value : UINT := DatatypeLimits.UINT_MAX_VALUE;
	actual : TIME;
	converted : BOOL;
	equal : BOOL;
END_VAR
TEST('Check_UINT_TO_TIME_Max');

// @TEST-RUN
converted := TryConvert_UINT_TO_Destination(value, actual);
equal := actual = UINT_TO_TIME(value);

// @TEST-ASSERT
AssertTrue(Condition := equal, Message := 'Did not convert UINT to TIME correctly');
AssertTrue(Condition := converted, Message := 'Did not report UINT to TIME conversion was successful');

TEST_FINISHED();
END_METHOD

METHOD PUBLIC Check_UINT_TO_TOD_Min
VAR
	value : UINT := DatatypeLimits.UINT_MIN_VALUE;
	actual : TOD;
	converted : BOOL;
	equal : BOOL;
END_VAR
TEST('Check_UINT_TO_TOD_Min');

// @TEST-RUN
converted := TryConvert_UINT_TO_Destination(value, actual);
equal := actual = UINT_TO_TOD(value);

// @TEST-ASSERT
AssertTrue(Condition := equal, Message := 'Did not convert UINT to TOD correctly');
AssertTrue(Condition := converted, Message := 'Did not report UINT to TOD conversion was successful');

TEST_FINISHED();
END_METHOD

METHOD PUBLIC Check_UINT_TO_TOD_Max
VAR
	value : UINT := DatatypeLimits.UINT_MAX_VALUE;
	actual : TOD;
	converted : BOOL;
	equal : BOOL;
END_VAR
TEST('Check_UINT_TO_TOD_Max');

// @TEST-RUN
converted := TryConvert_UINT_TO_Destination(value, actual);
equal := actual = UINT_TO_TOD(value);

// @TEST-ASSERT
AssertTrue(Condition := equal, Message := 'Did not convert UINT to TOD correctly');
AssertTrue(Condition := converted, Message := 'Did not report UINT to TOD conversion was successful');

TEST_FINISHED();
END_METHOD

METHOD PUBLIC Check_UINT_TO_UDINT_Min
VAR
	value : UINT := DatatypeLimits.UINT_MIN_VALUE;
	actual : UDINT;
	converted : BOOL;
	equal : BOOL;
END_VAR
TEST('Check_UINT_TO_UDINT_Min');

// @TEST-RUN
converted := TryConvert_UINT_TO_Destination(value, actual);
equal := actual = UINT_TO_UDINT(value);

// @TEST-ASSERT
AssertTrue(Condition := equal, Message := 'Did not convert UINT to UDINT correctly');
AssertTrue(Condition := converted, Message := 'Did not report UINT to UDINT conversion was successful');

TEST_FINISHED();
END_METHOD

METHOD PUBLIC Check_UINT_TO_UDINT_Max
VAR
	value : UINT := DatatypeLimits.UINT_MAX_VALUE;
	actual : UDINT;
	converted : BOOL;
	equal : BOOL;
END_VAR
TEST('Check_UINT_TO_UDINT_Max');

// @TEST-RUN
converted := TryConvert_UINT_TO_Destination(value, actual);
equal := actual = UINT_TO_UDINT(value);

// @TEST-ASSERT
AssertTrue(Condition := equal, Message := 'Did not convert UINT to UDINT correctly');
AssertTrue(Condition := converted, Message := 'Did not report UINT to UDINT conversion was successful');

TEST_FINISHED();
END_METHOD

METHOD PUBLIC Check_UINT_TO_UINT_Min
VAR
	value : UINT := DatatypeLimits.UINT_MIN_VALUE;
	actual : UINT;
	converted : BOOL;
	equal : BOOL;
END_VAR
TEST('Check_UINT_TO_UINT_Min');

// @TEST-RUN
converted := TryConvert_UINT_TO_Destination(value, actual);
equal := actual = value;

// @TEST-ASSERT
AssertTrue(Condition := equal, Message := 'Did not convert UINT to UINT correctly');
AssertTrue(Condition := converted, Message := 'Did not report UINT to UINT conversion was successful');

TEST_FINISHED();
END_METHOD

METHOD PUBLIC Check_UINT_TO_UINT_Max
VAR
	value : UINT := DatatypeLimits.UINT_MAX_VALUE;
	actual : UINT;
	converted : BOOL;
	equal : BOOL;
END_VAR
TEST('Check_UINT_TO_UINT_Max');

// @TEST-RUN
converted := TryConvert_UINT_TO_Destination(value, actual);
equal := actual = value;

// @TEST-ASSERT
AssertTrue(Condition := equal, Message := 'Did not convert UINT to UINT correctly');
AssertTrue(Condition := converted, Message := 'Did not report UINT to UINT conversion was successful');

TEST_FINISHED();
END_METHOD

METHOD PUBLIC Check_UINT_TO_ULINT_Min
VAR
	value : UINT := DatatypeLimits.UINT_MIN_VALUE;
	actual : ULINT;
	converted : BOOL;
	equal : BOOL;
END_VAR
TEST('Check_UINT_TO_ULINT_Min');

// @TEST-RUN
converted := TryConvert_UINT_TO_Destination(value, actual);
equal := actual = UINT_TO_ULINT(value);

// @TEST-ASSERT
AssertTrue(Condition := equal, Message := 'Did not convert UINT to ULINT correctly');
AssertTrue(Condition := converted, Message := 'Did not report UINT to ULINT conversion was successful');

TEST_FINISHED();
END_METHOD

METHOD PUBLIC Check_UINT_TO_ULINT_Max
VAR
	value : UINT := DatatypeLimits.UINT_MAX_VALUE;
	actual : ULINT;
	converted : BOOL;
	equal : BOOL;
END_VAR
TEST('Check_UINT_TO_ULINT_Max');

// @TEST-RUN
converted := TryConvert_UINT_TO_Destination(value, actual);
equal := actual = UINT_TO_ULINT(value);

// @TEST-ASSERT
AssertTrue(Condition := equal, Message := 'Did not convert UINT to ULINT correctly');
AssertTrue(Condition := converted, Message := 'Did not report UINT to ULINT conversion was successful');

TEST_FINISHED();
END_METHOD

METHOD PUBLIC Check_UINT_TO_USINT_Min
VAR
	value : UINT := DatatypeLimits.UINT_MIN_VALUE;
	actual : USINT;
	converted : BOOL;
	equal : BOOL;
END_VAR
TEST('Check_UINT_TO_USINT_Min');

// @TEST-RUN
converted := TryConvert_UINT_TO_Destination(value, actual);
equal := actual = UINT_TO_USINT(value);

// @TEST-ASSERT
AssertTrue(Condition := equal, Message := 'Did not convert UINT to USINT correctly');
AssertTrue(Condition := converted, Message := 'Did not report UINT to USINT conversion was successful');

TEST_FINISHED();
END_METHOD

METHOD PUBLIC Check_UINT_TO_USINT_TooHigh
VAR
	value : UINT := DatatypeLimits.UINT_MAX_VALUE;
	actual : USINT;
	converted : BOOL;
END_VAR
TEST('Check_UINT_TO_USINT_TooHigh');

// @TEST-RUN
converted := TryConvert_UINT_TO_Destination(value, actual);

// @TEST-ASSERT
AssertFalse(Condition := converted, Message := 'Did not report UINT to USINT conversion was prevented');

TEST_FINISHED();
END_METHOD

METHOD PUBLIC Check_UINT_TO_USINT_Max
VAR
	value : UINT := DatatypeLimits.MAX_VALUE_OF_UINT_WHICH_CAN_BE_HELD_IN_A_USINT;
	actual : USINT;
	converted : BOOL;
	equal : BOOL;
END_VAR
TEST('Check_UINT_TO_USINT_Max');

// @TEST-RUN
converted := TryConvert_UINT_TO_Destination(value, actual);
equal := actual = UINT_TO_USINT(value);

// @TEST-ASSERT
AssertTrue(Condition := equal, Message := 'Did not convert UINT to USINT correctly');
AssertTrue(Condition := converted, Message := 'Did not report UINT to USINT conversion was successful');

TEST_FINISHED();
END_METHOD

METHOD PUBLIC Check_UINT_TO_WORD_Min
VAR
	value : UINT := DatatypeLimits.UINT_MIN_VALUE;
	actual : WORD;
	converted : BOOL;
	equal : BOOL;
END_VAR
TEST('Check_UINT_TO_WORD_Min');

// @TEST-RUN
converted := TryConvert_UINT_TO_Destination(value, actual);
equal := actual = UINT_TO_WORD(value);

// @TEST-ASSERT
AssertTrue(Condition := equal, Message := 'Did not convert UINT to WORD correctly');
AssertTrue(Condition := converted, Message := 'Did not report UINT to WORD conversion was successful');

TEST_FINISHED();
END_METHOD

METHOD PUBLIC Check_UINT_TO_WORD_Max
VAR
	value : UINT := DatatypeLimits.UINT_MAX_VALUE;
	actual : WORD;
	converted : BOOL;
	equal : BOOL;
END_VAR
TEST('Check_UINT_TO_WORD_Max');

// @TEST-RUN
converted := TryConvert_UINT_TO_Destination(value, actual);
equal := actual = UINT_TO_WORD(value);

// @TEST-ASSERT
AssertTrue(Condition := equal, Message := 'Did not convert UINT to WORD correctly');
AssertTrue(Condition := converted, Message := 'Did not report UINT to WORD conversion was successful');

TEST_FINISHED();
END_METHOD

END_FUNCTION_BLOCK

// ---- Tests/UDINT_TO_TestSuite.TcPOU
FUNCTION_BLOCK PUBLIC UDINT_TO_TestSuite EXTENDS TcUnit.FB_TestSuite
VAR
END_VAR

Check_UDINT_TO_BOOL_Max();
Check_UDINT_TO_BOOL_Min();
Check_UDINT_TO_BYTE_Max();
Check_UDINT_TO_BYTE_Min();
Check_UDINT_TO_BYTE_TooHigh();
Check_UDINT_TO_WORD_Max();
Check_UDINT_TO_WORD_Min();
Check_UDINT_TO_WORD_TooHigh();
Check_UDINT_TO_DWORD_Max();
Check_UDINT_TO_DWORD_Min();
Check_UDINT_TO_LWORD_Max();
Check_UDINT_TO_LWORD_Min();
Check_UDINT_TO_SINT_Max();
Check_UDINT_TO_SINT_Min();
Check_UDINT_TO_SINT_TooHigh();
Check_UDINT_TO_INT_Max();
Check_UDINT_TO_INT_Min();
Check_UDINT_TO_INT_TooHigh();
Check_UDINT_TO_DINT_Max();
Check_UDINT_TO_DINT_Min();
Check_UDINT_TO_DINT_TooHigh();
Check_UDINT_TO_LINT_Max();
Check_UDINT_TO_LINT_Min();
Check_UDINT_TO_USINT_Max();
Check_UDINT_TO_USINT_Min();
Check_UDINT_TO_USINT_TooHigh();
Check_UDINT_TO_UINT_Max();
Check_UDINT_TO_UINT_Min();
Check_UDINT_TO_UINT_TooHigh();
Check_UDINT_TO_UDINT_Max();
Check_UDINT_TO_UDINT_Min();
Check_UDINT_TO_ULINT_Max();
Check_UDINT_TO_ULINT_Min();
Check_UDINT_TO_REAL_Max();
Check_UDINT_TO_REAL_Min();
Check_UDINT_TO_LREAL_Max();
Check_UDINT_TO_LREAL_Min();
Check_UDINT_TO_TIME_Max();
Check_UDINT_TO_TIME_Min();
Check_UDINT_TO_TOD_Max();
Check_UDINT_TO_TOD_Min();
Check_UDINT_TO_TOD_TooHigh();
Check_UDINT_TO_DATE_Max();
Check_UDINT_TO_DATE_Min();
Check_UDINT_TO_DT_Max();
Check_UDINT_TO_DT_Min();
Check_UDINT_TO_STRING_Max();
Check_UDINT_TO_STRING_Min();

METHOD PUBLIC Check_UDINT_TO_BOOL_Min
VAR
	value : UDINT := DatatypeLimits.UDINT_MIN_VALUE;
	actual : BOOL;
	converted : BOOL;
	equal : BOOL;
END_VAR
TEST('Check_UDINT_TO_BOOL_Min');

